// TwinCAT 3 PLC project Galimberti
// ProgramVersion: 3.1.4022.1
// libraries:
//   Tc2_MC2, * (Beckhoff Automation GmbH)
//   Tc2_MC2_Drive, * (Beckhoff Automation GmbH)
//   Tc2_Standard, * (Beckhoff Automation GmbH)
//   Tc2_System, * (Beckhoff Automation GmbH)
//   Tc3_Module, * (Beckhoff Automation GmbH)
// project tree:
//   DUTs/EVACUAZIONE SCARTI/ ES_ACTVAL.TcDUT, ES_MPO1.TcDUT, ES_PERSISTENT.TcDUT, ES_M.TcDUT, ES_ALARM.TcDUT, ES_S1.TcDUT, ES_S1PO1.TcDUT, ES_S2.TcDUT, ES_SEMAFORO.TcDUT, ES_T1.TcDUT, ES_T3.TcDUT, ES_T5.TcDUT, ES_T6.TcDUT
//   DUTs/RULLI_CENTRO_TAGLI/ dut_Axe_Status.TcDUT, dut_Dati_Pezzo.TcDUT
//   GVLs/EVACUAZIONE_SCARTI/ GVL_ES_IO.TcGVL
//   GVLs/RULLI CENTRO TAGLI/ GVL_CT_IO.TcGVL
//   / PlcTask.TcTTO, RulliCentroTagliTask.TcTTO
//   POUs/EVACUAZIONE_SCARTI/ EVACUAZIONE_SCARTI.TcPOU, MAIN.TcPOU
//   POUs/EVACUAZIONE_SCARTI/FB/ FB_AnalogSensor_full.TcPOU, FB_MMSensor_full.TcPOU, FB_Semaforo.TcPOU, fun_AreaM_SPEGNITUTTO.TcPOU
//   POUs/RULLI_CENTRO_TAGLI/FB/ FB_In_Position.TcPOU
//   POUs/RULLI_CENTRO_TAGLI/ MAIN_RCT.TcPOU, RULLI_CENTRO_TAGLI.TcPOU (not stored)
// real-time tasks:
//   TASK PlcTask: cycle T#10ms, priority 20, ADS port 350
//   TASK RulliCentroTagliTask: cycle T#10ms, priority 21, ADS port 351
// motion (NC):
//   TASK NC-Task 1 SAF: cycle T#2ms, priority 4, ADS port 501
//   TASK NC-Task 1 SVB: cycle T#10ms, priority 8, ADS port 511
//   AXIS C2M1 (id 1) // Motore catena 2
//     Dynamic: AccelerationMaximum=7500, DecelerationMaximum=7500, Acceleration=632.095593828125, Deceleration=632.095593828125, Jerk=1896.28678148437
//     Velo: RefSearch=4.21397062552083, RefSync=4.21397062552083, SlowManual=21.0698531276042, FastManual=126.419118765625, Fast=421.397062552083, Maximum=421.397062552083
//     OtherSettings: AllowMotionCmdToSlave=true
//     encoder EncType=8
//       EncPara: ScaleFactorNumerator=4.8964, ScaleFactorDenominator=1048576, MaxCount=#xffffffff
//     drive DrvType=9
//       DrvPara: MaxCount=#xffffffff, DriveControlDWord=#x00030100
//         Analog: VeloReferenz=463.536768807292, VeloScale=1.02400649589962, ScaleFactorActTorque=0.1
//         TimeComp: TaskDelayCycles=1
//     controller CtrType=1
//       CtrPara: PriorControlFactor=1
//         PosDiffControl: Range=30, Time=1
//         PID: PosKp=1.5
//         Observer: BandWidth=20
//   AXIS R1M1 (id 2) // Motore rulliera 1
//     Dynamic: Acceleration=1173.61, Deceleration=1173.61, Jerk=3520.84
//     Velo: RefSearch=7.8240862486901, RefSync=7.8240862486901, SlowManual=39.1204312434505, FastManual=234.722587460703, Fast=782.40862486901, Maximum=782.409
//     OtherSettings: AllowMotionCmdToSlave=true
//     encoder EncType=8
//       EncPara: ScaleFactorNumerator=9.091154, ScaleFactorDenominator=1048576, MaxCount=#xffffffff
//     drive DrvType=9
//       DrvPara: MaxCount=#xffffffff, DriveControlDWord=#x00030100
//         Analog: VeloReferenz=860.649487355912, VeloScale=1.02400649589962, ScaleFactorActTorque=0.1
//         TimeComp: TaskDelayCycles=1
//     controller CtrType=1
//       CtrPara: PriorControlFactor=1
//         Observer: BandWidth=20
//   AXIS C1M1 (id 3) // Motore sollevamento catenaria 1
//     Dynamic: Acceleration=194.243, Deceleration=194.243, Jerk=282.73
//     Velo: RefSearch=0.628289305598145, RefSync=0.628289305598145, SlowManual=3.14144652799072, FastManual=18.8486791679443, Fast=62.8289305598145, Maximum=62.8289
//     OtherSettings: AllowMotionCmdToSlave=true
//     encoder EncType=8
//       EncPara: ScaleFactorNumerator=1.15714, ScaleFactorDenominator=1048576, Inverse=true, MaxCount=#xffffffff
//         SoftEndMinControl: Enable=true, Range=590
//         SoftEndMaxControl: Enable=true, Range=1240
//     drive DrvType=9
//       DrvPara: Inverse=true, MaxCount=#xffffffff, DriveControlDWord=#x00030100
//         Analog: VeloReferenz=69.1118236157959, VeloScale=1.02400649589962, ScaleFactorActTorque=0.1
//         TimeComp: TaskDelayCycles=1
//     controller CtrType=1
//       CtrPara: PriorControlFactor=1
//         Observer: BandWidth=20
//   AXIS C1M3 (id 4) // Morore catenaria C1
//     Dynamic: AccelerationMaximum=7500, DecelerationMaximum=7500, Acceleration=900, Deceleration=900, Jerk=1896.28678148437
//     Velo: RefSearch=4.21397062552083, RefSync=4.21397062552083, SlowManual=21.0698531276042, FastManual=126.419118765625, Fast=421.397062552083, Maximum=421.397062552083
//     OtherSettings: AllowMotionCmdToSlave=true
//     encoder EncType=8
//       EncPara: ScaleFactorNumerator=4.8964, ScaleFactorDenominator=1048576, MaxCount=#xffffffff
//     drive DrvType=9
//       DrvPara: MaxCount=#xffffffff, DriveControlDWord=#x00030100
//         Analog: VeloReferenz=463.536768807292, VeloScale=1.02400649589962, ScaleFactorActTorque=0.1
//         TimeComp: TaskDelayCycles=1
//     controller CtrType=1
//       CtrPara: PriorControlFactor=1
//         PosDiffControl: Range=100, Time=1
//         PID: PosKp=2
//         Observer: BandWidth=20
//   AXIS C1M2 (id 5) // Rotazione catenaria C1
//     Dynamic: Acceleration=60.2372, Deceleration=60.2372, Jerk=180.712
//     Velo: RefSearch=0.401581141946615, RefSync=0.401581141946615, SlowManual=2.00790570973307, FastManual=12.0474342583984, Fast=40.1581141946615, Maximum=40.1581
//     OtherSettings: AllowMotionCmdToSlave=true
//     encoder EncType=8
//       EncPara: ScaleFactorNumerator=0.466615, ScaleFactorDenominator=1048576, MaxCount=#xffffffff
//     drive DrvType=9
//       DrvPara: MaxCount=#xffffffff, DriveControlDWord=#x00030100
//         Analog: VeloReferenz=44.1739256141276, VeloScale=1.02400649589962, ScaleFactorActTorque=0.1
//         TimeComp: TaskDelayCycles=1
//     controller CtrType=1
//       CtrPara: PriorControlFactor=1
//         Observer: BandWidth=20
//   AXIS C3 (id 6) // Catenaria 3
//     Dynamic: AccelerationMaximum=7000, Acceleration=689.378450181641, Deceleration=689.378450181641, Jerk=2068.13535054492
//     Velo: RefSearch=4.59585633454427, RefSync=4.59585633454427, SlowManual=22.9792816727214, FastManual=137.875690036328, Fast=459.585633454427, Maximum=459.585633454427
//     OtherSettings: AllowMotionCmdToSlave=true
//     encoder EncType=8
//       EncPara: ScaleFactorNumerator=5.34013, ScaleFactorDenominator=1048576, Inverse=true, MaxCount=#xffffffff
//     drive DrvType=9
//       DrvPara: Inverse=true, MaxCount=#xffffffff, DriveControlDWord=#x00030100
//         Analog: VeloReferenz=505.54419679987, VeloScale=1.02400649589962, ScaleFactorActTorque=0.1
//         TimeComp: TaskDelayCycles=1
//     controller CtrType=1
//       CtrPara: PriorControlFactor=1
//         Observer: BandWidth=20
//   AXIS C5 (id 7) // Catenaria 5
//     Dynamic: AccelerationMaximum=7000, Acceleration=689.378450181641, Deceleration=689.378450181641, Jerk=2068.13535054492
//     Velo: RefSearch=4.59585633454427, RefSync=4.59585633454427, SlowManual=22.9792816727214, FastManual=137.875690036328, Fast=459.585633454427, Maximum=459.585633454427
//     OtherSettings: AllowMotionCmdToSlave=true
//     encoder EncType=8
//       EncPara: ScaleFactorNumerator=5.34013, ScaleFactorDenominator=1048576, MaxCount=#xffffffff
//     drive DrvType=9
//       DrvPara: MaxCount=#xffffffff, DriveControlDWord=#x00030100
//         Analog: VeloReferenz=505.54419679987, VeloScale=1.02400649589962, ScaleFactorActTorque=0.1
//         TimeComp: TaskDelayCycles=1
//     controller CtrType=1
//       CtrPara: PriorControlFactor=1
//         Observer: BandWidth=20
//   AXIS C6 (id 8) // Catenaria 6
//     Dynamic: AccelerationMaximum=7000, Acceleration=689.378450181641, Deceleration=689.378450181641, Jerk=2068.13535054492
//     Velo: RefSearch=4.59585633454427, RefSync=4.59585633454427, SlowManual=22.9792816727214, FastManual=137.875690036328, Fast=459.585633454427, Maximum=459.585633454427
//     OtherSettings: AllowMotionCmdToSlave=true
//     encoder EncType=8
//       EncPara: ScaleFactorNumerator=5.34013, ScaleFactorDenominator=1048576, Inverse=true, MaxCount=#xffffffff
//     drive DrvType=9
//       DrvPara: Inverse=true, MaxCount=#xffffffff, DriveControlDWord=#x00030100
//         Analog: VeloReferenz=505.54419679987, VeloScale=1.02400649589962, ScaleFactorActTorque=0.1
//         TimeComp: TaskDelayCycles=1
//     controller CtrType=1
//       CtrPara: PriorControlFactor=1
//         Observer: BandWidth=20
//   AXIS R3 (id 9)
//     Dynamic: Acceleration=1353.648128, Deceleration=1353.648128, Jerk=4060.944384
//     Velo: RefSearch=9.02432085333333, RefSync=9.02432085333333, SlowManual=45.1216042666667, FastManual=270.7296256, Fast=902.432085333333, Maximum=902.432085333333
//     OtherSettings: AllowMotionCmdToSlave=true
//     encoder EncType=8
//       EncPara: ScaleFactorNumerator=10.48576, ScaleFactorDenominator=1048576, MaxCount=#xffffffff
//     drive DrvType=9
//       DrvPara: MaxCount=#xffffffff, DriveControlDWord=#x00030100
//         Analog: VeloReferenz=992.675293866667, VeloScale=1.02400649589962, ScaleFactorActTorque=0.1
//         TimeComp: TaskDelayCycles=1
//     controller CtrType=1
//       CtrPara: PriorControlFactor=1
//         Observer: BandWidth=20
//   AXIS R2 (id 10) // Rulliera 2
//     Dynamic: Acceleration=1173.61293730352, Deceleration=1173.61293730352, Jerk=3520.83881191055
//     Velo: RefSearch=7.8240862486901, RefSync=7.8240862486901, SlowManual=39.1204312434505, FastManual=234.722587460703, Fast=782.40862486901, Maximum=782.40862486901
//     OtherSettings: AllowMotionCmdToSlave=true
//     encoder EncType=8
//       EncPara: ScaleFactorNumerator=9.091154, ScaleFactorDenominator=1048576, MaxCount=#xffffffff
//     drive DrvType=9
//       DrvPara: MaxCount=#xffffffff, DriveControlDWord=#x00030100
//         Analog: VeloReferenz=860.649487355912, VeloScale=1.02400649589962, ScaleFactorActTorque=0.1
//         TimeComp: TaskDelayCycles=1
//     controller CtrType=1
//       CtrPara: PriorControlFactor=1
//         Observer: BandWidth=20
//   AXIS C4 (id 11)
//     Dynamic: AccelerationMaximum=7000, Acceleration=689.378450181641, Deceleration=689.378450181641, Jerk=2068.13535054492
//     Velo: RefSearch=4.59585633454427, RefSync=4.59585633454427, SlowManual=22.9792816727214, FastManual=137.875690036328, Fast=459.585633454427, Maximum=459.585633454427
//     OtherSettings: AllowMotionCmdToSlave=true
//     encoder EncType=8
//       EncPara: ScaleFactorNumerator=5.34013, ScaleFactorDenominator=1048576, MaxCount=#xffffffff
//     drive DrvType=9
//       DrvPara: MaxCount=#xffffffff, DriveControlDWord=#x00030100
//         Analog: VeloReferenz=505.54419679987, VeloScale=1.02400649589962, ScaleFactorActTorque=0.1
//         TimeComp: TaskDelayCycles=1
//     controller CtrType=1
//       CtrPara: PriorControlFactor=1
//         Observer: BandWidth=20
// I/O:
//   DEVICE Device 1 (EtherCAT), AmsNetId 192.168.30.180.2.1
//     Term 1 (EK1200) H-Q3 [EK1200-5000 EtherCAT Power supply (2A E-Bus)]
//       Term 2 (EL1008) [EL1008 8Ch. Dig. Input 24V, 3ms]
//       Term 3 (EL2008) [EL2008 8Ch. Dig. Output 24V, 0.5A]
//       Term 4 (EL6910) [EL6910, TwinSAFE PLC]
//       Term 5 (EK1110) [EK1110 EtherCAT extension]
//     Term 6 (EK1100) H-Q1 [EK1100 EtherCAT Coupler (2A E-Bus)]
//       Term 7 (EL1008) [EL1008 8Ch. Dig. Input 24V, 3ms]
//       Term 8 (EL1008) [EL1008 8Ch. Dig. Input 24V, 3ms]
//       Term 9 (EL2008) [EL2008 8Ch. Dig. Output 24V, 0.5A]
//       Term 10 (EL2008) [EL2008 8Ch. Dig. Output 24V, 0.5A]
//       Term 11 (EL3012) [EL3012 2Ch. Ana. Input 0-20mA DIFF]
//       Term 12 (EL3012) [EL3012 2Ch. Ana. Input 0-20mA DIFF]
//       Term 13 (EL2904) [EL2904, 4 Ch. Safety Output 24V, 0.5A, TwinSAFE]
//         modules: Module 1 (FSOES), Module 2 (DO)
//       Term 14 (EL2904) [EL2904, 4 Ch. Safety Output 24V, 0.5A, TwinSAFE]
//         modules: Module 1 (FSOES), Module 2 (DO)
//       Term 35 (EL6695) [EL6695 EtherCAT Bridge terminal (Primary)]
//       Term 15 (EK1110) [EK1110 EtherCAT extension]
//     Box 16 (EP6228-0022) M-CS1 [EP6228-0022 (IO Link Master)]
//       modules: Module 0 (DeviceState Inputs Device), Module 0 (DeviceState Inputs), Module 3 (IO-Link Slave) T1_SO1, Module 4 (empty), Module 5 (empty), Module 6 (empty), Module 7 (empty), Module 8 (empty), Module 9 (empty), Module 10 (empty)
//     Box 17 (EP6228-0022) T3-C01 [EP6228-0022 (IO Link Master)]
//       modules: Module 0 (DeviceState Inputs Device), Module 0 (DeviceState Inputs), Module 3 (IO-Link Slave), Module 2 (IO-Link Slave) S1_SO2, Module 3 (IO-Link Slave) S1_PO1, Module 6 (empty), Module 5 (IO-Link Slave) S1_Se1, Module 8 (empty), Module 7 (IO-Link Slave) T5_S1, Module 8 (IO-Link Slave) T5_SO1
//     Box 18 (EP1908) FS1 [EP1908, 8 Ch. Safety Input 24V, TwinSAFE]
//       modules: Module 1 (FSOE)
//     Term 39 (EK1100) [EK1100 EtherCAT Coupler (2A E-Bus)]
//       Term 40 (EL1008) [EL1008 8Ch. Dig. Input 24V, 3ms]
//       Term 41 (EL2008) [EL2008 8Ch. Dig. Output 24V, 0.5A]
//       Term 42 (EL2904) [EL2904, 4 Ch. Safety Output 24V, 0.5A, TwinSAFE]
//         modules: Module 1 (FSOES), Module 2 (DO)
//       Term 43 (EL1904) [EL1904, 4 Ch. Safety Input 24V, TwinSAFE]
//         modules: Module 1 (FSOES)
//       Term 44 (EL1904) [EL1904, 4 Ch. Safety Input 24V, TwinSAFE]
//         modules: Module 1 (FSOES)
//       Term 45 (EL1904) [EL1904, 4 Ch. Safety Input 24V, TwinSAFE]
//         modules: Module 1 (FSOES)
//       Term 46 (EK1122) [EK1122 2 port EtherCAT junction]
//         Box 47 (EP1008-0022) C1_CD4 [EP1008-0022 8 Ch. Dig. Input 24V, 3ms, M12]
//         Box 48 (EP6224-2022) C1_CO2 [EP6224-2022 (IO Link Master)]
//           modules: Module 1 (DeviceState Inputs Device), Module 2 (DeviceState Inputs), Module 3 (IO-Link Slave), Module 4 (IO-Link Slave), Module 5 (empty), Module 6 (empty)
//         Box 49 (EP1008-0022) C1_CD3 [EP1008-0022 8 Ch. Dig. Input 24V, 3ms, M12]
//         Box 50 (EP6224-2022) C1_CO1 [EP6224-2022 (IO Link Master)]
//           modules: Module 1 (DeviceState Inputs Device), Module 2 (DeviceState Inputs), Module 3 (IO-Link Slave), Module 4 (IO-Link Slave), Module 5 (IO-Link Slave), Module 6 (IO-Link Slave)
//         Box 51 (EP1008-0022) C1_CD2 [EP1008-0022 8 Ch. Dig. Input 24V, 3ms, M12]
//         Box 52 (EP1008-0022) C1_CD1 [EP1008-0022 8 Ch. Dig. Input 24V, 3ms, M12]
//         Box 53 (EP1008-0022) C2_CD4 [EP1008-0022 8 Ch. Dig. Input 24V, 3ms, M12]
//         Box 54 (EP6228-0022) C2_CO1 [EP6228-0022 (IO Link Master)]
//           modules: Module 1 (DeviceState Inputs Device), Module 2 (DeviceState Inputs), Module 3 (IO-Link Slave), Module 4 (IO-Link Slave), Module 5 (IO-Link Slave), Module 6 (IO-Link Slave), Module 7 (IO-Link Slave), Module 8 (IO-Link Slave), Module 9 (IO-Link Slave) - R1P5, Module 10 (IO-Link Slave) - R1P6
//         Box 55 (EP1008-0022) C2_CD3 [EP1008-0022 8 Ch. Dig. Input 24V, 3ms, M12]
//         Box 56 (EP1008-0022) C2_CD2 [EP1008-0022 8 Ch. Dig. Input 24V, 3ms, M12]
//         Box 57 (EP1008-0022) C2_CD1 [EP1008-0022 8 Ch. Dig. Input 24V, 3ms, M12]
//         Box 58 (EP6228-0022) C2_CO2 [EP6228-0022 (IO Link Master)]
//           modules: Module 1 (DeviceState Inputs Device), Module 2 (DeviceState Inputs), Module 3 (empty), Module 4 (IO-Link Slave) C1P1, Module 5 (empty), Module 6 (IO-Link Slave) R1P1, Module 7 (IO-Link Slave) R1P2, Module 8 (IO-Link Slave) R1P3, Module 9 (IO-Link Slave) R1P4, Module 10 (IO-Link Slave)
//         Box 59 (EP1908) C2_CS1 [EP1908, 8 Ch. Safety Input 24V, TwinSAFE]
//           modules: Module 1 (FSOE)
//         Box 60 (EP1908) C2_CS2 [EP1908, 8 Ch. Safety Input 24V, TwinSAFE]
//           modules: Module 1 (FSOE)
//       Term 61 (EK1122) [EK1122 2 port EtherCAT junction]
//         Drive 62 (AX5206-0000-0203) R2-C4 [AX5206-0000-0203 EtherCAT Drive (SoE, 2 Ch.)]
//         Drive 63 (AX5206-0000-0203) C3-R3 [AX5206-0000-0203 EtherCAT Drive (SoE, 2 Ch.)]
//         Drive 64 (AX5206-0000-0203) C5-C6 [AX5206-0000-0203 EtherCAT Drive (SoE, 2 Ch.)]
//         Drive 65 (AX5206-0000-0203) C1M2-C1M3 [AX5206-0000-0203 EtherCAT Drive (SoE, 2 Ch.)]
//         Drive 66 (AX5206-0000-0203) C2M1-R1M1 [AX5206-0000-0203 EtherCAT Drive (SoE, 2 Ch.)]
//         Drive 67 (AX5206-0000-0203) C1M1 [AX5112-0000-0203 EtherCAT Drive (SoE, 1 Ch.)]
//         Box 68 (S100) R1M2 [S100]
//         Box 99 (S100) R2 [S100]
//         Box 100 (S100) R3 [S100]
//         Box 101 (EP6228-0022) C5_CO1 [EP6228-0022 (IO Link Master)]
//           modules: Module 1 (DeviceState Inputs Device), Module 2 (DeviceState Inputs), Module 3 (IO-Link Slave), Module 4 (IO-Link Slave), Module 5 (IO-Link Slave), Module 6 (empty), Module 7 (IO-Link Slave), Module 8 (IO-Link Slave), Module 9 (IO-Link Slave), Module 10 (empty)
//         Box 102 (EP1008-0022) C5_CD1 [EP1008-0022 8 Ch. Dig. Input 24V, 3ms, M12]
//         Box 103 (EP1908) C5_CS1 [EP1908, 8 Ch. Safety Input 24V, TwinSAFE]
//           modules: Module 1 (FSOE)
//         Box 104 (EP6228-0022) C5_CO2 [EP6228-0022 (IO Link Master)]
//           modules: Module 1 (DeviceState Inputs Device), Module 2 (DeviceState Inputs), Module 3 (IO-Link Slave), Module 4 (IO-Link Slave), Module 5 (IO-Link Slave), Module 6 (IO-Link Slave), Module 7 (IO-Link Slave), Module 8 (IO-Link Slave), Module 9 (IO-Link Slave), Module 10 (IO-Link Slave)
//         Box 105 (EP1008-0022) C5_CD2 [EP1008-0022 8 Ch. Dig. Input 24V, 3ms, M12]
//         Box 106 (EP1008-0022) C5_CD3 [EP1008-0022 8 Ch. Dig. Input 24V, 3ms, M12]
//         Box 115 (EP1008-0022) C3CD1 [EP1008-0022 8 Ch. Dig. Input 24V, 3ms, M12]
//         Box 116 (EP6228-0022) C3CO1 [EP6228-0022 (IO Link Master)]
//           modules: Module 1 (DeviceState Inputs Device), Module 2 (DeviceState Inputs), Module 3 (empty), Module 4 (IO-Link Slave), Module 5 (IO-Link Slave), Module 6 (empty), Module 7 (empty), Module 8 (IO-Link Slave), Module 9 (IO-Link Slave), Module 10 (IO-Link Slave)
//         Box 117 (EP1008-0022) C3CD2 [EP1008-0022 8 Ch. Dig. Input 24V, 3ms, M12]
//         Box 118 (EP1908) C3CS1 [EP1908, 8 Ch. Safety Input 24V, TwinSAFE]
//           modules: Module 1 (FSOE)
//   DEVICE Device 4 (RT-Ethernet Protocol) (disabled), AmsNetId 192.168.30.180.5.1
//   DEVICE Device 5 (NOV-DP-RAM) (disabled)
// variable links:
//   Device 1 (EtherCAT) <-> Device 1 (EtherCAT)/Box 18 (EP1908) FS1
//     Term 1 (EK1200) H-Q3/Term 4 (EL6910)/ConnectionOutputs/TwinSafeGroup_ES.Box 18 (EP1908) - Module 1 (FSOE)_10 RxPDO <-> Module 1 (FSOE)/FSOE Inputs/FSOE
//   Device 1 (EtherCAT) <-> Device 1 (EtherCAT)/Term 1 (EK1200) H-Q3/Term 4 (EL6910)
//     Box 18 (EP1908) FS1/Module 1 (FSOE)/FSOE Outputs/FSOE <-> ConnectionInputs/TwinSafeGroup_ES.Box 18 (EP1908) - Module 1 (FSOE)_10 TxPDO
//     Term 39 (EK1100)/Term 42 (EL2904)/Module 1 (FSOES)/TxPDO/FSOE <-> ConnectionOutputs/TwinSafeGroup_ES.Term 42 (EL2904) - Module 1 (FSOES)_31 RxPDO
//     Term 39 (EK1100)/Term 44 (EL1904)/Module 1 (FSOES)/TxPDO/FSOE <-> ConnectionOutputs/TwinSafeGroup_ES.Term 44 (EL1904) - Module 1 (FSOES)_33 RxPDO
//     Term 39 (EK1100)/Term 43 (EL1904)/Module 1 (FSOES)/RxPDO/FSOE <-> ConnectionInputs/TwinSafeGroup_ES.Term 43 (EL1904) - Module 1 (FSOES)_32 TxPDO
//     Term 39 (EK1100)/Term 44 (EL1904)/Module 1 (FSOES)/RxPDO/FSOE <-> ConnectionInputs/TwinSafeGroup_ES.Term 44 (EL1904) - Module 1 (FSOES)_33 TxPDO
//     Term 39 (EK1100)/Term 46 (EK1122)/Box 59 (EP1908) C2_CS1/Module 1 (FSOE)/FSOE Inputs/FSOE <-> ConnectionOutputs/TwinSafeGroup_ES.Box 59 (EP1908) C2_CS1 - Module 1 (FSOE)_35 RxPDO
//     Term 39 (EK1100)/Term 46 (EK1122)/Box 60 (EP1908) C2_CS2/Module 1 (FSOE)/FSOE Inputs/FSOE <-> ConnectionOutputs/TwinSafeGroup_ES.Box 60 (EP1908) C2_CS2 - Module 1 (FSOE)_36 RxPDO
//     Term 39 (EK1100)/Term 46 (EK1122)/Box 59 (EP1908) C2_CS1/Module 1 (FSOE)/FSOE Outputs/FSOE <-> ConnectionInputs/TwinSafeGroup_ES.Box 59 (EP1908) C2_CS1 - Module 1 (FSOE)_35 TxPDO
//     Term 39 (EK1100)/Term 61 (EK1122)/Box 118 (EP1908) C3CS1/Module 1 (FSOE)/FSOE Inputs/FSOE <-> ConnectionOutputs/TwinSafeGroup_ES.Box 118 (EP1908) C3CS1 - Module 1 (FSOE)_39 RxPDO
//     Term 39 (EK1100)/Term 61 (EK1122)/Box 118 (EP1908) C3CS1/Module 1 (FSOE)/FSOE Outputs/FSOE <-> ConnectionInputs/TwinSafeGroup_ES.Box 118 (EP1908) C3CS1 - Module 1 (FSOE)_39 TxPDO
//     Term 6 (EK1100) H-Q1/Term 13 (EL2904)/Module 1 (FSOES)/TxPDO/FSOE <-> ConnectionOutputs/TwinSafeGroup_ES.Term 13 (EL2904) - Module 1 (FSOES)_8 RxPDO
//   Device 1 (EtherCAT) <-> Device 1 (EtherCAT)/Term 39 (EK1100)/Term 42 (EL2904)
//     Term 1 (EK1200) H-Q3/Term 4 (EL6910)/ConnectionInputs/TwinSafeGroup_ES.Term 42 (EL2904) - Module 1 (FSOES)_31 TxPDO <-> Module 1 (FSOES)/RxPDO/FSOE
//   Device 1 (EtherCAT) <-> Device 1 (EtherCAT)/Term 39 (EK1100)/Term 43 (EL1904)
//     Term 1 (EK1200) H-Q3/Term 4 (EL6910)/ConnectionOutputs/TwinSafeGroup_ES.Term 43 (EL1904) - Module 1 (FSOES)_32 RxPDO <-> Module 1 (FSOES)/TxPDO/FSOE
//   Device 1 (EtherCAT) <-> Device 1 (EtherCAT)/Term 39 (EK1100)/Term 45 (EL1904)
//     Term 1 (EK1200) H-Q3/Term 4 (EL6910)/ConnectionInputs/TwinSafeGroup_ES.Term 45 (EL1904) - Module 1 (FSOES)_34 TxPDO <-> Module 1 (FSOES)/RxPDO/FSOE
//     Term 1 (EK1200) H-Q3/Term 4 (EL6910)/ConnectionOutputs/TwinSafeGroup_ES.Term 45 (EL1904) - Module 1 (FSOES)_34 RxPDO <-> Module 1 (FSOES)/TxPDO/FSOE
//   Device 1 (EtherCAT) <-> Device 1 (EtherCAT)/Term 39 (EK1100)/Term 46 (EK1122)/Box 60 (EP1908) C2_CS2
//     Term 1 (EK1200) H-Q3/Term 4 (EL6910)/ConnectionInputs/TwinSafeGroup_ES.Box 60 (EP1908) C2_CS2 - Module 1 (FSOE)_36 TxPDO <-> Module 1 (FSOE)/FSOE Outputs/FSOE
//   Device 1 (EtherCAT) <-> Device 1 (EtherCAT)/Term 39 (EK1100)/Term 61 (EK1122)/Box 103 (EP1908) C5_CS1
//     Term 1 (EK1200) H-Q3/Term 4 (EL6910)/ConnectionInputs/TwinSafeGroup_ES.Box 103 (EP1908) C5_CS1 - Module 1 (FSOE)_40 TxPDO <-> Module 1 (FSOE)/FSOE Outputs/FSOE
//     Term 1 (EK1200) H-Q3/Term 4 (EL6910)/ConnectionOutputs/TwinSafeGroup_ES.Box 103 (EP1908) C5_CS1 - Module 1 (FSOE)_40 RxPDO <-> Module 1 (FSOE)/FSOE Inputs/FSOE
//   Device 1 (EtherCAT) <-> Device 1 (EtherCAT)/Term 6 (EK1100) H-Q1/Term 13 (EL2904)
//     Term 1 (EK1200) H-Q3/Term 4 (EL6910)/ConnectionInputs/TwinSafeGroup_ES.Term 13 (EL2904) - Module 1 (FSOES)_8 TxPDO <-> Module 1 (FSOES)/RxPDO/FSOE
//   NC-Task 1 SAF/Axes/C1M1 <-> Device 1 (EtherCAT)/Term 39 (EK1100)/Term 61 (EK1122)/Drive 67 (AX5206-0000-0203) C1M1
//     Drive/Inputs/In/nDataIn1 <-> AT/Following distance
//     Drive/Inputs/In/nDcOutputTime <-> InfoData/DcOutputShift
//     Drive/Inputs/In/nState1 <-> AT/Drive status word @bit 8
//     Drive/Inputs/In/nState2 <-> AT/Drive status word
//     Drive/Inputs/In/nState4 @bit 1 <-> WcState/InputToggle
//     Drive/Inputs/In/nState4 <-> WcState/WcState
//     Drive/Outputs/Out/nCtrl1 <-> MDT/Master control word @bit 8
//     Drive/Outputs/Out/nDataOut1 <-> MDT/Position command value
//     Enc/Inputs/In/nDataIn1 <-> AT/Position feedback 1 value
//     Enc/Inputs/In/nDcInputTime <-> InfoData/DcInputShift
//     Enc/Inputs/In/nState4 @bit 1 <-> WcState/InputToggle
//     Enc/Inputs/In/nState4 <-> WcState/WcState
//   NC-Task 1 SAF/Axes/C1M2 <-> Device 1 (EtherCAT)/Term 39 (EK1100)/Term 61 (EK1122)/Drive 65 (AX5206-0000-0203) C1M2-C1M3
//     Drive/Inputs/In/nDataIn1 <-> AT 1/Following distance
//     Drive/Inputs/In/nDataIn3[0] <-> AT 1/Torque feedback value
//     Drive/Inputs/In/nDcOutputTime <-> InfoData/DcOutputShift
//     Drive/Inputs/In/nState1 <-> AT 1/Drive status word @bit 8
//     Drive/Inputs/In/nState2 <-> AT 1/Drive status word
//     Drive/Inputs/In/nState4 @bit 1 <-> WcState/InputToggle
//     Drive/Inputs/In/nState4 <-> WcState/WcState
//     Drive/Outputs/Out/nCtrl1 <-> MDT 1/Master control word @bit 8
//     Drive/Outputs/Out/nDataOut1 <-> MDT 1/Position command value
//     Enc/Inputs/In/nDataIn1 <-> AT 1/Position feedback 1 value
//     Enc/Inputs/In/nDcInputTime <-> InfoData/DcInputShift
//     Enc/Inputs/In/nState4 @bit 1 <-> WcState/InputToggle
//     Enc/Inputs/In/nState4 <-> WcState/WcState
//   NC-Task 1 SAF/Axes/C1M3 <-> Device 1 (EtherCAT)/Term 39 (EK1100)/Term 61 (EK1122)/Drive 65 (AX5206-0000-0203) C1M2-C1M3
//     Drive/Inputs/In/nDataIn1 <-> AT 2/Following distance
//     Drive/Inputs/In/nDcOutputTime <-> InfoData/DcOutputShift
//     Drive/Inputs/In/nState1 <-> AT 2/Drive status word @bit 8
//     Drive/Inputs/In/nState2 <-> AT 2/Drive status word
//     Drive/Inputs/In/nState4 @bit 1 <-> WcState/InputToggle
//     Drive/Inputs/In/nState4 <-> WcState/WcState
//     Drive/Outputs/Out/nCtrl1 <-> MDT 2/Master control word @bit 8
//     Drive/Outputs/Out/nDataOut1 <-> MDT 2/Position command value
//     Enc/Inputs/In/nDataIn1 <-> AT 2/Position feedback 1 value
//     Enc/Inputs/In/nDcInputTime <-> InfoData/DcInputShift
//     Enc/Inputs/In/nState4 @bit 1 <-> WcState/InputToggle
//     Enc/Inputs/In/nState4 <-> WcState/WcState
//   NC-Task 1 SAF/Axes/C2M1 <-> Device 1 (EtherCAT)/Term 39 (EK1100)/Term 61 (EK1122)/Drive 66 (AX5206-0000-0203) C2M1-R1M1
//     Drive/Inputs/In/nDataIn1 <-> AT 1/Following distance
//     Drive/Inputs/In/nDcOutputTime <-> InfoData/DcOutputShift
//     Drive/Inputs/In/nState1 <-> AT 1/Drive status word @bit 8
//     Drive/Inputs/In/nState2 <-> AT 1/Drive status word
//     Drive/Inputs/In/nState4 @bit 1 <-> WcState/InputToggle
//     Drive/Inputs/In/nState4 <-> WcState/WcState
//     Drive/Outputs/Out/nCtrl1 <-> MDT 1/Master control word @bit 8
//     Drive/Outputs/Out/nDataOut1 <-> MDT 1/Position command value
//     Enc/Inputs/In/nDataIn1 <-> AT 1/Position feedback 1 value
//     Enc/Inputs/In/nDcInputTime <-> InfoData/DcInputShift
//     Enc/Inputs/In/nState4 @bit 1 <-> WcState/InputToggle
//     Enc/Inputs/In/nState4 <-> WcState/WcState
//   NC-Task 1 SAF/Axes/C3 <-> Device 1 (EtherCAT)/Term 39 (EK1100)/Term 61 (EK1122)/Drive 63 (AX5206-0000-0203) C3-R3
//     Drive/Inputs/In/nDataIn1 <-> AT 1/Following distance
//     Drive/Inputs/In/nDcOutputTime <-> InfoData/DcOutputShift
//     Drive/Inputs/In/nState1 <-> AT 1/Drive status word @bit 8
//     Drive/Inputs/In/nState2 <-> AT 1/Drive status word
//     Drive/Inputs/In/nState4 @bit 1 <-> WcState/InputToggle
//     Drive/Inputs/In/nState4 <-> WcState/WcState
//     Drive/Outputs/Out/nCtrl1 <-> MDT 1/Master control word @bit 8
//     Drive/Outputs/Out/nDataOut1 <-> MDT 1/Position command value
//     Enc/Inputs/In/nDataIn1 <-> AT 1/Position feedback 1 value
//     Enc/Inputs/In/nDcInputTime <-> InfoData/DcInputShift
//     Enc/Inputs/In/nState4 @bit 1 <-> WcState/InputToggle
//     Enc/Inputs/In/nState4 <-> WcState/WcState
//   NC-Task 1 SAF/Axes/C4 <-> Device 1 (EtherCAT)/Term 39 (EK1100)/Term 61 (EK1122)/Drive 62 (AX5206-0000-0203) R2-C4
//     Drive/Inputs/In/nDataIn1 <-> AT 2/Following distance
//     Drive/Inputs/In/nDcOutputTime <-> InfoData/DcOutputShift
//     Drive/Inputs/In/nState1 <-> AT 2/Drive status word @bit 8
//     Drive/Inputs/In/nState2 <-> AT 2/Drive status word
//     Drive/Inputs/In/nState4 @bit 1 <-> WcState/InputToggle
//     Drive/Inputs/In/nState4 <-> WcState/WcState
//     Drive/Outputs/Out/nCtrl1 <-> MDT 2/Master control word @bit 8
//     Drive/Outputs/Out/nDataOut1 <-> MDT 2/Position command value
//     Enc/Inputs/In/nDataIn1 <-> AT 2/Position feedback 1 value
//     Enc/Inputs/In/nDcInputTime <-> InfoData/DcInputShift
//     Enc/Inputs/In/nState4 @bit 1 <-> WcState/InputToggle
//     Enc/Inputs/In/nState4 <-> WcState/WcState
//   NC-Task 1 SAF/Axes/C5 <-> Device 1 (EtherCAT)/Term 39 (EK1100)/Term 61 (EK1122)/Drive 64 (AX5206-0000-0203) C5-C6
//     Drive/Inputs/In/nDataIn1 <-> AT 1/Following distance
//     Drive/Inputs/In/nDcOutputTime <-> InfoData/DcOutputShift
//     Drive/Inputs/In/nState1 <-> AT 1/Drive status word @bit 8
//     Drive/Inputs/In/nState2 <-> AT 1/Drive status word
//     Drive/Inputs/In/nState4 @bit 1 <-> WcState/InputToggle
//     Drive/Inputs/In/nState4 <-> WcState/WcState
//     Drive/Outputs/Out/nCtrl1 <-> MDT 1/Master control word @bit 8
//     Drive/Outputs/Out/nDataOut1 <-> MDT 1/Position command value
//     Enc/Inputs/In/nDataIn1 <-> AT 1/Position feedback 1 value
//     Enc/Inputs/In/nDcInputTime <-> InfoData/DcInputShift
//     Enc/Inputs/In/nState4 @bit 1 <-> WcState/InputToggle
//     Enc/Inputs/In/nState4 <-> WcState/WcState
//   NC-Task 1 SAF/Axes/C6 <-> Device 1 (EtherCAT)/Term 39 (EK1100)/Term 61 (EK1122)/Drive 64 (AX5206-0000-0203) C5-C6
//     Drive/Inputs/In/nDataIn1 <-> AT 2/Following distance
//     Drive/Inputs/In/nDcOutputTime <-> InfoData/DcOutputShift
//     Drive/Inputs/In/nState1 <-> AT 2/Drive status word @bit 8
//     Drive/Inputs/In/nState2 <-> AT 2/Drive status word
//     Drive/Inputs/In/nState4 @bit 1 <-> WcState/InputToggle
//     Drive/Inputs/In/nState4 <-> WcState/WcState
//     Drive/Outputs/Out/nCtrl1 <-> MDT 2/Master control word @bit 8
//     Drive/Outputs/Out/nDataOut1 <-> MDT 2/Position command value
//     Enc/Inputs/In/nDataIn1 <-> AT 2/Position feedback 1 value
//     Enc/Inputs/In/nDcInputTime <-> InfoData/DcInputShift
//     Enc/Inputs/In/nState4 @bit 1 <-> WcState/InputToggle
//     Enc/Inputs/In/nState4 <-> WcState/WcState
//   NC-Task 1 SAF/Axes/R1M1 <-> Device 1 (EtherCAT)/Term 39 (EK1100)/Term 61 (EK1122)/Drive 66 (AX5206-0000-0203) C2M1-R1M1
//     Drive/Inputs/In/nDataIn1 <-> AT 2/Following distance
//     Drive/Inputs/In/nDcOutputTime <-> InfoData/DcOutputShift
//     Drive/Inputs/In/nState1 <-> AT 2/Drive status word @bit 8
//     Drive/Inputs/In/nState2 <-> AT 2/Drive status word
//     Drive/Inputs/In/nState4 @bit 1 <-> WcState/InputToggle
//     Drive/Inputs/In/nState4 <-> WcState/WcState
//     Drive/Outputs/Out/nCtrl1 <-> MDT 2/Master control word @bit 8
//     Drive/Outputs/Out/nDataOut1 <-> MDT 2/Position command value
//     Enc/Inputs/In/nDataIn1 <-> AT 2/Position feedback 1 value
//     Enc/Inputs/In/nDcInputTime <-> InfoData/DcInputShift
//     Enc/Inputs/In/nState4 @bit 1 <-> WcState/InputToggle
//     Enc/Inputs/In/nState4 <-> WcState/WcState
//   NC-Task 1 SAF/Axes/R2 <-> Device 1 (EtherCAT)/Term 39 (EK1100)/Term 61 (EK1122)/Drive 62 (AX5206-0000-0203) R2-C4
//     Drive/Inputs/In/nDataIn1 <-> AT 1/Following distance
//     Drive/Inputs/In/nDcOutputTime <-> InfoData/DcOutputShift
//     Drive/Inputs/In/nState1 <-> AT 1/Drive status word @bit 8
//     Drive/Inputs/In/nState2 <-> AT 1/Drive status word
//     Drive/Inputs/In/nState4 @bit 1 <-> WcState/InputToggle
//     Drive/Inputs/In/nState4 <-> WcState/WcState
//     Drive/Outputs/Out/nCtrl1 <-> MDT 1/Master control word @bit 8
//     Drive/Outputs/Out/nDataOut1 <-> MDT 1/Position command value
//     Enc/Inputs/In/nDataIn1 <-> AT 1/Position feedback 1 value
//     Enc/Inputs/In/nDcInputTime <-> InfoData/DcInputShift
//     Enc/Inputs/In/nState4 @bit 1 <-> WcState/InputToggle
//     Enc/Inputs/In/nState4 <-> WcState/WcState
//   NC-Task 1 SAF/Axes/R3 <-> Device 1 (EtherCAT)/Term 39 (EK1100)/Term 61 (EK1122)/Drive 63 (AX5206-0000-0203) C3-R3
//     Drive/Inputs/In/nDataIn1 <-> AT 2/Following distance
//     Drive/Inputs/In/nDcOutputTime <-> InfoData/DcOutputShift
//     Drive/Inputs/In/nState1 <-> AT 2/Drive status word @bit 8
//     Drive/Inputs/In/nState2 <-> AT 2/Drive status word
//     Drive/Inputs/In/nState4 @bit 1 <-> WcState/InputToggle
//     Drive/Inputs/In/nState4 <-> WcState/WcState
//     Drive/Outputs/Out/nCtrl1 <-> MDT 2/Master control word @bit 8
//     Drive/Outputs/Out/nDataOut1 <-> MDT 2/Position command value
//     Enc/Inputs/In/nDataIn1 <-> AT 2/Position feedback 1 value
//     Enc/Inputs/In/nDcInputTime <-> InfoData/DcInputShift
//     Enc/Inputs/In/nState4 @bit 1 <-> WcState/InputToggle
//     Enc/Inputs/In/nState4 <-> WcState/WcState
//   Galimberti/Galimberti Instance <-> Device 1 (EtherCAT)/Box 16 (EP6228-0022) M-CS1
//     PlcTask Inputs/.glo_analog_in_MCS1[1] <-> Module 3 (IO-Link Slave) T1_SO1/IO-Link Port1/Distance
//     RulliCentroTagliTask Inputs/.glo_IOLState_MCS1[{1..8}] <-> Module 0 (DeviceState Inputs)/DeviceState Inputs/State Ch{1..8}  (8 links)
//     RulliCentroTagliTask Inputs/.glo_State_MCS1[1] <-> InfoData/State
//     RulliCentroTagliTask Inputs/.glo_WcState_MCS1[1] <-> WcState/WcState
//   Galimberti/Galimberti Instance <-> Device 1 (EtherCAT)/Box 17 (EP6228-0022) T3-C01
//     PlcTask Inputs/.glo_analog_in_T3C01[1] <-> Module 2 (IO-Link Slave) S1_SO2/IO-Link Port2/PDV1
//     PlcTask Inputs/.glo_analog_in_T3C01[2] <-> Module 8 (IO-Link Slave) T5_SO1/IO-Link Port8/PDV1
//     PlcTask Inputs/.glo_dig_in_T3C01[10] <-> Module 3 (IO-Link Slave)/IO-Link Port1/Port1: process data
//     PlcTask Inputs/.glo_dig_in_T3C01[1] <-> Module 3 (IO-Link Slave) S1_PO1/IO-Link Port3_in/Switchstate Pin 1 (Bit0.0)
//     PlcTask Inputs/.glo_dig_in_T3C01[2] <-> Module 3 (IO-Link Slave) S1_PO1/IO-Link Port3_in/Switchstate Pin 2 (Bit0.1)
//     PlcTask Inputs/.glo_dig_in_T3C01[3] <-> Module 3 (IO-Link Slave) S1_PO1/IO-Link Port3_in/Switchstate Pin 3 (Bit0.2)
//     PlcTask Inputs/.glo_dig_in_T3C01[4] <-> Module 3 (IO-Link Slave) S1_PO1/IO-Link Port3_in/Switchstate Pin 4 (Bit0.3)
//     PlcTask Inputs/.glo_dig_in_T3C01[5] <-> Module 3 (IO-Link Slave) S1_PO1/IO-Link Port3_in/Switchstate Pin 5 (Bit0.4)
//     PlcTask Inputs/.glo_dig_in_T3C01[6] <-> Module 3 (IO-Link Slave) S1_PO1/IO-Link Port3_in/Switchstate Pin 6 (Bit0.5)
//     PlcTask Inputs/.glo_dig_in_T3C01[7] <-> Module 3 (IO-Link Slave) S1_PO1/IO-Link Port3_in/Switchstate Pin 7 (Bit0.6)
//     PlcTask Inputs/.glo_dig_in_T3C01[8] <-> Module 3 (IO-Link Slave) S1_PO1/IO-Link Port3_in/Switchstate Pin 8 (Bit0.7)
//     PlcTask Inputs/.glo_dig_in_T3C01[25] <-> Module 7 (IO-Link Slave) T5_S1/IO-Link Port7/Port7: process data
//     PlcTask Outputs/.S1_Se1.analog{0..5} <-> Module 5 (IO-Link Slave) S1_Se1/IO-Link Port5/Port5: process data[{0..5}]  (6 links)
//     PlcTask Outputs/.glo_dig_out_T3C01[1] <-> Module 3 (IO-Link Slave) S1_PO1/IO-Link Port3_out/Switchstate Pin 1 (Bit0.0)
//     PlcTask Outputs/.glo_dig_out_T3C01[2] <-> Module 3 (IO-Link Slave) S1_PO1/IO-Link Port3_out/Switchstate Pin 2 (Bit0.1)
//     PlcTask Outputs/.glo_dig_out_T3C01[3] <-> Module 3 (IO-Link Slave) S1_PO1/IO-Link Port3_out/Switchstate Pin 3 (Bit0.2)
//     PlcTask Outputs/.glo_dig_out_T3C01[4] <-> Module 3 (IO-Link Slave) S1_PO1/IO-Link Port3_out/Switchstate Pin 4 (Bit0.3)
//     PlcTask Outputs/.glo_dig_out_T3C01[5] <-> Module 3 (IO-Link Slave) S1_PO1/IO-Link Port3_out/Switchstate Pin 5 (Bit0.4)
//     PlcTask Outputs/.glo_dig_out_T3C01[6] <-> Module 3 (IO-Link Slave) S1_PO1/IO-Link Port3_out/Switchstate Pin 6 (Bit0.5)
//     PlcTask Outputs/.glo_dig_out_T3C01[7] <-> Module 3 (IO-Link Slave) S1_PO1/IO-Link Port3_out/Switchstate Pin 7 (Bit0.6)
//     PlcTask Outputs/.glo_dig_out_T3C01[8] <-> Module 3 (IO-Link Slave) S1_PO1/IO-Link Port3_out/Switchstate Pin 8 (Bit0.7)
//     RulliCentroTagliTask Inputs/.glo_IOLState_T3C01[1] <-> Module 0 (DeviceState Inputs)/DeviceState Inputs/State Ch1
//     RulliCentroTagliTask Inputs/.glo_IOLState_T3C01[2] <-> Module 0 (DeviceState Inputs)/DeviceState Inputs/State Ch2
//     RulliCentroTagliTask Inputs/.glo_IOLState_T3C01[3] <-> Module 0 (DeviceState Inputs)/DeviceState Inputs/State Ch3
//     RulliCentroTagliTask Inputs/.glo_IOLState_T3C01[4] <-> Module 0 (DeviceState Inputs)/DeviceState Inputs/State Ch4
//     RulliCentroTagliTask Inputs/.glo_IOLState_T3C01[5] <-> Module 0 (DeviceState Inputs)/DeviceState Inputs/State Ch5
//     RulliCentroTagliTask Inputs/.glo_IOLState_T3C01[6] <-> Module 0 (DeviceState Inputs)/DeviceState Inputs/State Ch6
//     RulliCentroTagliTask Inputs/.glo_IOLState_T3C01[7] <-> Module 0 (DeviceState Inputs)/DeviceState Inputs/State Ch7
//     RulliCentroTagliTask Inputs/.glo_IOLState_T3C01[8] <-> Module 0 (DeviceState Inputs)/DeviceState Inputs/State Ch8
//     RulliCentroTagliTask Inputs/.glo_State_T3C01[1] <-> InfoData/State
//     RulliCentroTagliTask Inputs/.glo_WcState_T3C01[1] <-> WcState/WcState
//   Galimberti/Galimberti Instance <-> Device 1 (EtherCAT)/Term 1 (EK1200) H-Q3/Term 2 (EL1008)
//     RulliCentroTagliTask Inputs/.glo_State_HQ3[1] <-> InfoData/State
//     RulliCentroTagliTask Inputs/.glo_WcState_HQ3[1] <-> WcState/WcState
//     RulliCentroTagliTask Inputs/.glo_dig_in_HQ3[{1..8}] <-> Channel {1..8}/Input  (8 links)
//   Galimberti/Galimberti Instance <-> Device 1 (EtherCAT)/Term 1 (EK1200) H-Q3/Term 3 (EL2008)
//     RulliCentroTagliTask Inputs/.glo_State_HQ3[2] <-> InfoData/State
//     RulliCentroTagliTask Inputs/.glo_WcState_HQ3[2] <-> WcState/WcState
//     RulliCentroTagliTask Outputs/.glo_dig_out_HQ3[{1..8}] <-> Channel {1..8}/Output  (8 links)
//   Galimberti/Galimberti Instance <-> Device 1 (EtherCAT)/Term 1 (EK1200) H-Q3/Term 4 (EL6910)
//     PlcTask Inputs/.TS_AreaM_ON <-> StandardInputs/TwinSafeGroup_ES.toTC_AreaM_ON_23
//     PlcTask Inputs/.TS_AreaS_ON <-> StandardInputs/TwinSafeGroup_ES.toTC_AreaS_ON_24
//     PlcTask Outputs/.TS_ErrAck <-> StandardOutputs/TwinSafeGroup_ES.ErrorAcknowledgement_1
//     PlcTask Outputs/.TS_MPO1_Rst_Area_Macinatore <-> StandardOutputs/TwinSafeGroup_ES.fromTC_Rst_Area_Macinatore_43
//     PlcTask Outputs/.TS_Run_GrpES <-> StandardOutputs/TwinSafeGroup_ES.Run_2
//     PlcTask Outputs/.TS_S1PO1_btn_R <-> StandardOutputs/TwinSafeGroup_ES.fromTC_S1PO1_RestartE_stop_20
//     RulliCentroTagliTask Inputs/.TS_AreaM_OFF <-> StandardInputs/TwinSafeGroup_ES.toTC_AreaM_ON_23
//     RulliCentroTagliTask Inputs/.TS_ComErr <-> StandardInputs/TwinSafeGroup_ES.toTC_ComErr_27
//     RulliCentroTagliTask Inputs/.TS_FBErr <-> StandardInputs/TwinSafeGroup_ES.toTC_FBErr_28
//     RulliCentroTagliTask Inputs/.TS_R1P1_Pls_Eme <-> StandardInputs/TwinSafeGroup_ES.toTC_Eme_Ok_38
//     RulliCentroTagliTask Inputs/.TS_S1PO1_btn_Emerg <-> StandardInputs/TwinSafeGroup_ES.toTC_S1PO1_Emergency_21
//     RulliCentroTagliTask Inputs/.TS_S1PR1_Door <-> StandardInputs/TwinSafeGroup_ES.toTC_S1PR1_Door_22
//     RulliCentroTagliTask Inputs/.glo_State_HQ3[3] <-> InfoData/State
//     RulliCentroTagliTask Inputs/.glo_WcState_HQ3[3] <-> WcState/WcState
//     RulliCentroTagliTask Inputs/.glo_dig_in_BOX18[{1..8}] <-> Connection Info Data/TwinSafeGroup_ES.Box 18 (EP1908) - Module 1 (FSOE)_10 Info Data/Input Safe Data InputChannel{1..8}  (8 links)
//     RulliCentroTagliTask Inputs/.glo_dig_in_C2_CS1[1] <-> Connection Info Data/TwinSafeGroup_ES.Box 59 (EP1908) C2_CS1 - Module 1 (FSOE)_35 Info Data/Input Safe Data InputChannel1
//     RulliCentroTagliTask Inputs/.glo_dig_in_C2_CS1[2] <-> Connection Info Data/TwinSafeGroup_ES.Box 59 (EP1908) C2_CS1 - Module 1 (FSOE)_35 Info Data/Input Safe Data InputChannel2
//     RulliCentroTagliTask Inputs/.glo_dig_in_C2_CS1[3] <-> Connection Info Data/TwinSafeGroup_ES.Box 59 (EP1908) C2_CS1 - Module 1 (FSOE)_35 Info Data/Input Safe Data InputChannel3
//     RulliCentroTagliTask Inputs/.glo_dig_in_C2_CS1[4] <-> Connection Info Data/TwinSafeGroup_ES.Box 59 (EP1908) C2_CS1 - Module 1 (FSOE)_35 Info Data/Input Safe Data InputChannel4
//     RulliCentroTagliTask Inputs/.glo_dig_in_C2_CS1[5] <-> Connection Info Data/TwinSafeGroup_ES.Box 59 (EP1908) C2_CS1 - Module 1 (FSOE)_35 Info Data/Input Safe Data InputChannel5
//     RulliCentroTagliTask Inputs/.glo_dig_in_C2_CS1[6] <-> Connection Info Data/TwinSafeGroup_ES.Box 59 (EP1908) C2_CS1 - Module 1 (FSOE)_35 Info Data/Input Safe Data InputChannel6
//     RulliCentroTagliTask Inputs/.glo_dig_in_C2_CS1[7] <-> Connection Info Data/TwinSafeGroup_ES.Box 59 (EP1908) C2_CS1 - Module 1 (FSOE)_35 Info Data/Input Safe Data InputChannel7
//     RulliCentroTagliTask Inputs/.glo_dig_in_C2_CS1[8] <-> Connection Info Data/TwinSafeGroup_ES.Box 59 (EP1908) C2_CS1 - Module 1 (FSOE)_35 Info Data/Input Safe Data InputChannel8
//     RulliCentroTagliTask Inputs/.glo_dig_in_C2_CS2[1] <-> Connection Info Data/TwinSafeGroup_ES.Box 60 (EP1908) C2_CS2 - Module 1 (FSOE)_36 Info Data/Input Safe Data InputChannel1
//     RulliCentroTagliTask Inputs/.glo_dig_in_C2_CS2[2] <-> Connection Info Data/TwinSafeGroup_ES.Box 60 (EP1908) C2_CS2 - Module 1 (FSOE)_36 Info Data/Input Safe Data InputChannel2
//     RulliCentroTagliTask Inputs/.glo_dig_in_C2_CS2[3] <-> Connection Info Data/TwinSafeGroup_ES.Box 60 (EP1908) C2_CS2 - Module 1 (FSOE)_36 Info Data/Input Safe Data InputChannel3
//     RulliCentroTagliTask Inputs/.glo_dig_in_C2_CS2[4] <-> Connection Info Data/TwinSafeGroup_ES.Box 60 (EP1908) C2_CS2 - Module 1 (FSOE)_36 Info Data/Input Safe Data InputChannel4
//     RulliCentroTagliTask Inputs/.glo_dig_in_C2_CS2[5] <-> Connection Info Data/TwinSafeGroup_ES.Box 60 (EP1908) C2_CS2 - Module 1 (FSOE)_36 Info Data/Input Safe Data InputChannel5
//     RulliCentroTagliTask Inputs/.glo_dig_in_C2_CS2[6] <-> Connection Info Data/TwinSafeGroup_ES.Box 60 (EP1908) C2_CS2 - Module 1 (FSOE)_36 Info Data/Input Safe Data InputChannel6
//     RulliCentroTagliTask Inputs/.glo_dig_in_C2_CS2[7] <-> Connection Info Data/TwinSafeGroup_ES.Box 60 (EP1908) C2_CS2 - Module 1 (FSOE)_36 Info Data/Input Safe Data InputChannel7
//     RulliCentroTagliTask Inputs/.glo_dig_in_C2_CS2[8] <-> Connection Info Data/TwinSafeGroup_ES.Box 60 (EP1908) C2_CS2 - Module 1 (FSOE)_36 Info Data/Input Safe Data InputChannel8
//     RulliCentroTagliTask Inputs/.glo_dig_in_C5_CS1[1] <-> Connection Info Data/TwinSafeGroup_ES.Box 103 (EP1908) C5_CS1 - Module 1 (FSOE)_40 Info Data/Input Safe Data InputChannel1
//     RulliCentroTagliTask Inputs/.glo_dig_in_C5_CS1[2] <-> Connection Info Data/TwinSafeGroup_ES.Box 103 (EP1908) C5_CS1 - Module 1 (FSOE)_40 Info Data/Input Safe Data InputChannel2
//     RulliCentroTagliTask Inputs/.glo_dig_in_C5_CS1[3] <-> Connection Info Data/TwinSafeGroup_ES.Box 103 (EP1908) C5_CS1 - Module 1 (FSOE)_40 Info Data/Input Safe Data InputChannel3
//     RulliCentroTagliTask Inputs/.glo_dig_in_C5_CS1[4] <-> Connection Info Data/TwinSafeGroup_ES.Box 103 (EP1908) C5_CS1 - Module 1 (FSOE)_40 Info Data/Input Safe Data InputChannel4
//     RulliCentroTagliTask Inputs/.glo_dig_in_C5_CS1[5] <-> Connection Info Data/TwinSafeGroup_ES.Box 103 (EP1908) C5_CS1 - Module 1 (FSOE)_40 Info Data/Input Safe Data InputChannel5
//     RulliCentroTagliTask Inputs/.glo_dig_in_C5_CS1[6] <-> Connection Info Data/TwinSafeGroup_ES.Box 103 (EP1908) C5_CS1 - Module 1 (FSOE)_40 Info Data/Input Safe Data InputChannel6
//     RulliCentroTagliTask Inputs/.glo_dig_in_C5_CS1[7] <-> Connection Info Data/TwinSafeGroup_ES.Box 103 (EP1908) C5_CS1 - Module 1 (FSOE)_40 Info Data/Input Safe Data InputChannel7
//     RulliCentroTagliTask Inputs/.glo_dig_in_C5_CS1[8] <-> Connection Info Data/TwinSafeGroup_ES.Box 103 (EP1908) C5_CS1 - Module 1 (FSOE)_40 Info Data/Input Safe Data InputChannel8
//     RulliCentroTagliTask Inputs/.glo_dig_in_C3_CS1[{1..8}] <-> Connection Info Data/TwinSafeGroup_ES.Box 118 (EP1908) C3CS1 - Module 1 (FSOE)_39 Info Data/Input Safe Data InputChannel{1..8}  (8 links)
//     RulliCentroTagliTask Outputs/.TS_R1P1_Reset_Eme <-> StandardOutputs/TwinSafeGroup_ES.fromTC_R1P1_RestartE_Stop_RCS_41
//     RulliCentroTagliTask Outputs/.TS_R1P1_Reset_Eme_2 <-> StandardOutputs/TwinSafeGroup_ES.fromTC_R1P1_RestartE_Stop_RCS2_42
//   Galimberti/Galimberti Instance <-> Device 1 (EtherCAT)/Term 1 (EK1200) H-Q3/Term 5 (EK1110)
//     RulliCentroTagliTask Inputs/.glo_State_HQ3[4] <-> InfoData/State
//   Galimberti/Galimberti Instance <-> Device 1 (EtherCAT)/Term 39 (EK1100)/Term 40 (EL1008)
//     RulliCentroTagliTask Inputs/.glo_dig_in_Term_40[{1..8}] <-> Channel {1..8}/Input  (8 links)
//   Galimberti/Galimberti Instance <-> Device 1 (EtherCAT)/Term 39 (EK1100)/Term 46 (EK1122)/Box 47 (EP1008-0022) C1_CD4
//     RulliCentroTagliTask Inputs/.glo_State_C1CD4[1] <-> InfoData/State
//     RulliCentroTagliTask Inputs/.glo_WcState_C1CD4[1] <-> WcState/WcState
//     RulliCentroTagliTask Inputs/.glo_dig_in_C1CD4[{1..8}] <-> Channel {1..8}/Input  (8 links)
//   Galimberti/Galimberti Instance <-> Device 1 (EtherCAT)/Term 39 (EK1100)/Term 46 (EK1122)/Box 48 (EP6224-2022) C1_CO2
//     RulliCentroTagliTask Outputs/.glo_dig_out_C1CO2[1] <-> Module 3 (IO-Link Slave)/IO-Link Port1/Port1: process data
//     RulliCentroTagliTask Outputs/.glo_dig_out_C1CO2[2] <-> Module 4 (IO-Link Slave)/IO-Link Port2/Port2: process data
//   Galimberti/Galimberti Instance <-> Device 1 (EtherCAT)/Term 39 (EK1100)/Term 46 (EK1122)/Box 49 (EP1008-0022) C1_CD3
//     RulliCentroTagliTask Inputs/.glo_dig_in_C1CD3[{1..8}] <-> Channel {1..8}/Input  (8 links)
//   Galimberti/Galimberti Instance <-> Device 1 (EtherCAT)/Term 39 (EK1100)/Term 46 (EK1122)/Box 50 (EP6224-2022) C1_CO1
//     RulliCentroTagliTask Outputs/.glo_dig_out_C1CO1[{1..4}] <-> Module {3..6} (IO-Link Slave)/IO-Link Port{1..4}/Port{1..4}: process data  (4 links)
//   Galimberti/Galimberti Instance <-> Device 1 (EtherCAT)/Term 39 (EK1100)/Term 46 (EK1122)/Box 51 (EP1008-0022) C1_CD2
//     RulliCentroTagliTask Inputs/.glo_dig_in_C1CD2[{1..8}] <-> Channel {1..8}/Input  (8 links)
//   Galimberti/Galimberti Instance <-> Device 1 (EtherCAT)/Term 39 (EK1100)/Term 46 (EK1122)/Box 52 (EP1008-0022) C1_CD1
//     RulliCentroTagliTask Inputs/.glo_dig_in_C1CD1[{1..8}] <-> Channel {1..8}/Input  (8 links)
//   Galimberti/Galimberti Instance <-> Device 1 (EtherCAT)/Term 39 (EK1100)/Term 46 (EK1122)/Box 53 (EP1008-0022) C2_CD4
//     RulliCentroTagliTask Inputs/.glo_State_C2CD4[1] <-> InfoData/State
//     RulliCentroTagliTask Inputs/.glo_WcState_C2CD4[1] <-> WcState/WcState
//     RulliCentroTagliTask Inputs/.glo_dig_in_C2CD4[{1..8}] <-> Channel {1..8}/Input  (8 links)
//   Galimberti/Galimberti Instance <-> Device 1 (EtherCAT)/Term 39 (EK1100)/Term 46 (EK1122)/Box 54 (EP6228-0022) C2_CO1
//     RulliCentroTagliTask Inputs/.glo_dig_in_R1P5[1] <-> Module 9 (IO-Link Slave) - R1P5/IO-Link Port7_in/Switchstate Pin 1 (Bit0.0)
//     RulliCentroTagliTask Inputs/.glo_dig_in_R1P5[2] <-> Module 9 (IO-Link Slave) - R1P5/IO-Link Port7_in/Switchstate Pin 2 (Bit0.1)
//     RulliCentroTagliTask Inputs/.glo_dig_in_R1P5[3] <-> Module 9 (IO-Link Slave) - R1P5/IO-Link Port7_in/Switchstate Pin 3 (Bit0.2)
//     RulliCentroTagliTask Inputs/.glo_dig_in_R1P5[4] <-> Module 9 (IO-Link Slave) - R1P5/IO-Link Port7_in/Switchstate Pin 4 (Bit0.3)
//     RulliCentroTagliTask Inputs/.glo_dig_in_R1P5[5] <-> Module 9 (IO-Link Slave) - R1P5/IO-Link Port7_in/Switchstate Pin 5 (Bit0.4)
//     RulliCentroTagliTask Inputs/.glo_dig_in_R1P5[6] <-> Module 9 (IO-Link Slave) - R1P5/IO-Link Port7_in/Switchstate Pin 6 (Bit0.5)
//     RulliCentroTagliTask Inputs/.glo_dig_in_R1P5[7] <-> Module 9 (IO-Link Slave) - R1P5/IO-Link Port7_in/Switchstate Pin 7 (Bit0.6)
//     RulliCentroTagliTask Inputs/.glo_dig_in_R1P5[8] <-> Module 9 (IO-Link Slave) - R1P5/IO-Link Port7_in/Switchstate Pin 8 (Bit0.7)
//     RulliCentroTagliTask Inputs/.glo_dig_in_R1P6[1] <-> Module 10 (IO-Link Slave) - R1P6/IO-Link Port8_in/Switchstate Pin 1 (Bit0.0)
//     RulliCentroTagliTask Inputs/.glo_dig_in_R1P6[2] <-> Module 10 (IO-Link Slave) - R1P6/IO-Link Port8_in/Switchstate Pin 2 (Bit0.1)
//     RulliCentroTagliTask Inputs/.glo_dig_in_R1P6[3] <-> Module 10 (IO-Link Slave) - R1P6/IO-Link Port8_in/Switchstate Pin 3 (Bit0.2)
//     RulliCentroTagliTask Inputs/.glo_dig_in_R1P6[4] <-> Module 10 (IO-Link Slave) - R1P6/IO-Link Port8_in/Switchstate Pin 4 (Bit0.3)
//     RulliCentroTagliTask Inputs/.glo_dig_in_R1P6[5] <-> Module 10 (IO-Link Slave) - R1P6/IO-Link Port8_in/Switchstate Pin 5 (Bit0.4)
//     RulliCentroTagliTask Inputs/.glo_dig_in_R1P6[6] <-> Module 10 (IO-Link Slave) - R1P6/IO-Link Port8_in/Switchstate Pin 6 (Bit0.5)
//     RulliCentroTagliTask Inputs/.glo_dig_in_R1P6[7] <-> Module 10 (IO-Link Slave) - R1P6/IO-Link Port8_in/Switchstate Pin 7 (Bit0.6)
//     RulliCentroTagliTask Inputs/.glo_dig_in_R1P6[8] <-> Module 10 (IO-Link Slave) - R1P6/IO-Link Port8_in/Switchstate Pin 8 (Bit0.7)
//     RulliCentroTagliTask Outputs/.glo_dig_out_C2CO1[1] <-> Module 4 (IO-Link Slave)/IO-Link Port2/Port2: process data
//     RulliCentroTagliTask Outputs/.glo_dig_out_C2CO1[2] <-> Module 5 (IO-Link Slave)/IO-Link Port3/Port3: process data
//     RulliCentroTagliTask Outputs/.glo_dig_out_C2CO1[3] <-> Module 6 (IO-Link Slave)/IO-Link Port4/Port4: process data
//   Galimberti/Galimberti Instance <-> Device 1 (EtherCAT)/Term 39 (EK1100)/Term 46 (EK1122)/Box 55 (EP1008-0022) C2_CD3
//     RulliCentroTagliTask Inputs/.glo_dig_in_C2CD3[{1..8}] <-> Channel {1..8}/Input  (8 links)
//   Galimberti/Galimberti Instance <-> Device 1 (EtherCAT)/Term 39 (EK1100)/Term 46 (EK1122)/Box 56 (EP1008-0022) C2_CD2
//     RulliCentroTagliTask Inputs/.glo_dig_in_C2CD2[{1..8}] <-> Channel {1..8}/Input  (8 links)
//   Galimberti/Galimberti Instance <-> Device 1 (EtherCAT)/Term 39 (EK1100)/Term 46 (EK1122)/Box 57 (EP1008-0022) C2_CD1
//     RulliCentroTagliTask Inputs/.glo_dig_in_C2CD1[{1..8}] <-> Channel {1..8}/Input  (8 links)
//   Galimberti/Galimberti Instance <-> Device 1 (EtherCAT)/Term 39 (EK1100)/Term 46 (EK1122)/Box 58 (EP6228-0022) C2_CO2
//     RulliCentroTagliTask Inputs/.glo_IOLState_C2CO2[{1..8}] <-> Module 2 (DeviceState Inputs)/DeviceState Inputs/State Ch{1..8}  (8 links)
//     RulliCentroTagliTask Inputs/.glo_dig_in_C1P1[{1..8}] <-> Module 4 (IO-Link Slave) C1P1/IO-Link Port2_in/Switchstate Pin {1..8} (Bit0.{0..7})  (8 links)
//     RulliCentroTagliTask Inputs/.glo_dig_in_R1P1[1] <-> Module 6 (IO-Link Slave) R1P1/IO-Link Port4_in/Switchstate Pin 1 (Bit0.0)
//     RulliCentroTagliTask Inputs/.glo_dig_in_R1P1[2] <-> Module 6 (IO-Link Slave) R1P1/IO-Link Port4_in/Switchstate Pin 2 (Bit0.1)
//     RulliCentroTagliTask Inputs/.glo_dig_in_R1P1[3] <-> Module 6 (IO-Link Slave) R1P1/IO-Link Port4_in/Switchstate Pin 3 (Bit0.2)
//     RulliCentroTagliTask Inputs/.glo_dig_in_R1P1[4] <-> Module 6 (IO-Link Slave) R1P1/IO-Link Port4_in/Switchstate Pin 4 (Bit0.3)
//     RulliCentroTagliTask Inputs/.glo_dig_in_R1P1[5] <-> Module 6 (IO-Link Slave) R1P1/IO-Link Port4_in/Switchstate Pin 5 (Bit0.4)
//     RulliCentroTagliTask Inputs/.glo_dig_in_R1P1[6] <-> Module 6 (IO-Link Slave) R1P1/IO-Link Port4_in/Switchstate Pin 6 (Bit0.5)
//     RulliCentroTagliTask Inputs/.glo_dig_in_R1P1[7] <-> Module 6 (IO-Link Slave) R1P1/IO-Link Port4_in/Switchstate Pin 7 (Bit0.6)
//     RulliCentroTagliTask Inputs/.glo_dig_in_R1P1[8] <-> Module 6 (IO-Link Slave) R1P1/IO-Link Port4_in/Switchstate Pin 8 (Bit0.7)
//     RulliCentroTagliTask Inputs/.glo_dig_in_R1P1[9] <-> Module 6 (IO-Link Slave) R1P1/IO-Link Port4_in/Switchstate Pin 9 (Bit1.0)
//     RulliCentroTagliTask Inputs/.glo_dig_in_R1P2[1] <-> Module 7 (IO-Link Slave) R1P2/IO-Link Port5_in/Switchstate Pin 1 (Bit0.0)
//     RulliCentroTagliTask Inputs/.glo_dig_in_R1P2[2] <-> Module 7 (IO-Link Slave) R1P2/IO-Link Port5_in/Switchstate Pin 2 (Bit0.1)
//     RulliCentroTagliTask Inputs/.glo_dig_in_R1P2[3] <-> Module 7 (IO-Link Slave) R1P2/IO-Link Port5_in/Switchstate Pin 3 (Bit0.2)
//     RulliCentroTagliTask Inputs/.glo_dig_in_R1P2[4] <-> Module 7 (IO-Link Slave) R1P2/IO-Link Port5_in/Switchstate Pin 4 (Bit0.3)
//     RulliCentroTagliTask Inputs/.glo_dig_in_R1P2[5] <-> Module 7 (IO-Link Slave) R1P2/IO-Link Port5_in/Switchstate Pin 5 (Bit0.4)
//     RulliCentroTagliTask Inputs/.glo_dig_in_R1P2[6] <-> Module 7 (IO-Link Slave) R1P2/IO-Link Port5_in/Switchstate Pin 6 (Bit0.5)
//     RulliCentroTagliTask Inputs/.glo_dig_in_R1P2[7] <-> Module 7 (IO-Link Slave) R1P2/IO-Link Port5_in/Switchstate Pin 7 (Bit0.6)
//     RulliCentroTagliTask Inputs/.glo_dig_in_R1P2[8] <-> Module 7 (IO-Link Slave) R1P2/IO-Link Port5_in/Switchstate Pin 8 (Bit0.7)
//     RulliCentroTagliTask Inputs/.glo_dig_in_R1P3[1] <-> Module 8 (IO-Link Slave) R1P3/IO-Link Port6_in/Switchstate Pin 1 (Bit0.0)
//     RulliCentroTagliTask Inputs/.glo_dig_in_R1P3[2] <-> Module 8 (IO-Link Slave) R1P3/IO-Link Port6_in/Switchstate Pin 2 (Bit0.1)
//     RulliCentroTagliTask Inputs/.glo_dig_in_R1P3[3] <-> Module 8 (IO-Link Slave) R1P3/IO-Link Port6_in/Switchstate Pin 3 (Bit0.2)
//     RulliCentroTagliTask Inputs/.glo_dig_in_R1P3[4] <-> Module 8 (IO-Link Slave) R1P3/IO-Link Port6_in/Switchstate Pin 4 (Bit0.3)
//     RulliCentroTagliTask Inputs/.glo_dig_in_R1P3[5] <-> Module 8 (IO-Link Slave) R1P3/IO-Link Port6_in/Switchstate Pin 5 (Bit0.4)
//     RulliCentroTagliTask Inputs/.glo_dig_in_R1P3[6] <-> Module 8 (IO-Link Slave) R1P3/IO-Link Port6_in/Switchstate Pin 6 (Bit0.5)
//     RulliCentroTagliTask Inputs/.glo_dig_in_R1P3[7] <-> Module 8 (IO-Link Slave) R1P3/IO-Link Port6_in/Switchstate Pin 7 (Bit0.6)
//     RulliCentroTagliTask Inputs/.glo_dig_in_R1P3[8] <-> Module 8 (IO-Link Slave) R1P3/IO-Link Port6_in/Switchstate Pin 8 (Bit0.7)
//     RulliCentroTagliTask Inputs/.glo_dig_in_R1P4[1] <-> Module 9 (IO-Link Slave) R1P4/IO-Link Port7_in/Switchstate Pin 1 (Bit0.0)
//     RulliCentroTagliTask Inputs/.glo_dig_in_R1P4[2] <-> Module 9 (IO-Link Slave) R1P4/IO-Link Port7_in/Switchstate Pin 2 (Bit0.1)
//     RulliCentroTagliTask Inputs/.glo_dig_in_R1P4[3] <-> Module 9 (IO-Link Slave) R1P4/IO-Link Port7_in/Switchstate Pin 3 (Bit0.2)
//     RulliCentroTagliTask Inputs/.glo_dig_in_R1P4[4] <-> Module 9 (IO-Link Slave) R1P4/IO-Link Port7_in/Switchstate Pin 4 (Bit0.3)
//     RulliCentroTagliTask Inputs/.glo_dig_in_R1P4[5] <-> Module 9 (IO-Link Slave) R1P4/IO-Link Port7_in/Switchstate Pin 5 (Bit0.4)
//     RulliCentroTagliTask Inputs/.glo_dig_in_R1P4[6] <-> Module 9 (IO-Link Slave) R1P4/IO-Link Port7_in/Switchstate Pin 6 (Bit0.5)
//     RulliCentroTagliTask Inputs/.glo_dig_in_R1P4[7] <-> Module 9 (IO-Link Slave) R1P4/IO-Link Port7_in/Switchstate Pin 7 (Bit0.6)
//     RulliCentroTagliTask Inputs/.glo_dig_in_R1P4[8] <-> Module 9 (IO-Link Slave) R1P4/IO-Link Port7_in/Switchstate Pin 8 (Bit0.7)
//     RulliCentroTagliTask Outputs/.RCT_Semaforo.analog{0..5} <-> Module 10 (IO-Link Slave)/IO-Link Port8/Port8: process data[{0..5}]  (6 links)
//     RulliCentroTagliTask Outputs/.glo_dig_out_C1P1[{8..14}] <-> Module 4 (IO-Link Slave) C1P1/IO-Link Port2_out/Switchstate Pin {9..15} (Bit1.{0..6})  (7 links)
//     RulliCentroTagliTask Outputs/.glo_dig_out_R1P1[{10..16}] <-> Module 6 (IO-Link Slave) R1P1/IO-Link Port4_out/Switchstate Pin {10..16} (Bit1.{1..7})  (7 links)
//   Galimberti/Galimberti Instance <-> Device 1 (EtherCAT)/Term 39 (EK1100)/Term 61 (EK1122)/Box 100 (S100) R3
//     RulliCentroTagliTask Inputs/RULLI_CENTRO_TAGLI.R3_Inverter_Act_Alarm <-> Transmit PDO Mapping Parameter 3/subIndex 3
//     RulliCentroTagliTask Outputs/RULLI_CENTRO_TAGLI.R3_Inverter_Inverter_Cmd <-> Receive PDO Mapping Parameter 3/subIndex 2
//     RulliCentroTagliTask Outputs/RULLI_CENTRO_TAGLI.R3_Inverter_Speed_Override <-> Receive PDO Mapping Parameter 3/subIndex 1
//   Galimberti/Galimberti Instance <-> Device 1 (EtherCAT)/Term 39 (EK1100)/Term 61 (EK1122)/Box 101 (EP6228-0022) C5_CO1
//     RulliCentroTagliTask Outputs/.glo_dig_out_C5CO1[1] <-> Module 3 (IO-Link Slave)/IO-Link Port1/Port1: process data
//     RulliCentroTagliTask Outputs/.glo_dig_out_C5CO1[2] <-> Module 4 (IO-Link Slave)/IO-Link Port2/Port2: process data
//     RulliCentroTagliTask Outputs/.glo_dig_out_C5CO1[3] <-> Module 5 (IO-Link Slave)/IO-Link Port3/Port3: process data
//     RulliCentroTagliTask Outputs/.glo_dig_out_C5CO1[4] <-> Module 7 (IO-Link Slave)/IO-Link Port5/Port5: process data
//     RulliCentroTagliTask Outputs/.glo_dig_out_C5CO1[5] <-> Module 8 (IO-Link Slave)/IO-Link Port6/Port6: process data
//     RulliCentroTagliTask Outputs/.glo_dig_out_C5CO1[6] <-> Module 9 (IO-Link Slave)/IO-Link Port7/Port7: process data
//   Galimberti/Galimberti Instance <-> Device 1 (EtherCAT)/Term 39 (EK1100)/Term 61 (EK1122)/Box 102 (EP1008-0022) C5_CD1
//     RulliCentroTagliTask Inputs/.glo_dig_in_C5CD1[{1..8}] <-> Channel {1..8}/Input  (8 links)
//   Galimberti/Galimberti Instance <-> Device 1 (EtherCAT)/Term 39 (EK1100)/Term 61 (EK1122)/Box 104 (EP6228-0022) C5_CO2
//     RulliCentroTagliTask Inputs/.glo_dig_in_C5CO2[1] <-> Module 5 (IO-Link Slave)/IO-Link Port3/Port3: process data
//     RulliCentroTagliTask Inputs/.glo_dig_in_C5CO2[2] <-> Module 6 (IO-Link Slave)/IO-Link Port4/Port4: process data
//     RulliCentroTagliTask Inputs/.glo_dig_in_R3P1[1] <-> Module 7 (IO-Link Slave)/IO-Link Port5_in/Switchstate Pin 1 (Bit0.0)
//     RulliCentroTagliTask Inputs/.glo_dig_in_R3P1[2] <-> Module 7 (IO-Link Slave)/IO-Link Port5_in/Switchstate Pin 2 (Bit0.1)
//     RulliCentroTagliTask Inputs/.glo_dig_in_R3P1[3] <-> Module 7 (IO-Link Slave)/IO-Link Port5_in/Switchstate Pin 3 (Bit0.2)
//     RulliCentroTagliTask Inputs/.glo_dig_in_R3P1[4] <-> Module 7 (IO-Link Slave)/IO-Link Port5_in/Switchstate Pin 4 (Bit0.3)
//     RulliCentroTagliTask Inputs/.glo_dig_in_R3P1[5] <-> Module 7 (IO-Link Slave)/IO-Link Port5_in/Switchstate Pin 5 (Bit0.4)
//     RulliCentroTagliTask Inputs/.glo_dig_in_R3P1[6] <-> Module 7 (IO-Link Slave)/IO-Link Port5_in/Switchstate Pin 6 (Bit0.5)
//     RulliCentroTagliTask Inputs/.glo_dig_in_R3P1[7] <-> Module 7 (IO-Link Slave)/IO-Link Port5_in/Switchstate Pin 7 (Bit0.6)
//     RulliCentroTagliTask Inputs/.glo_dig_in_R3P1[8] <-> Module 7 (IO-Link Slave)/IO-Link Port5_in/Switchstate Pin 8 (Bit0.7)
//     RulliCentroTagliTask Inputs/.glo_dig_in_R3P2[1] <-> Module 8 (IO-Link Slave)/IO-Link Port6_in/Switchstate Pin 1 (Bit0.0)
//     RulliCentroTagliTask Inputs/.glo_dig_in_R3P2[2] <-> Module 8 (IO-Link Slave)/IO-Link Port6_in/Switchstate Pin 2 (Bit0.1)
//     RulliCentroTagliTask Inputs/.glo_dig_in_R3P2[3] <-> Module 8 (IO-Link Slave)/IO-Link Port6_in/Switchstate Pin 3 (Bit0.2)
//     RulliCentroTagliTask Inputs/.glo_dig_in_R3P2[4] <-> Module 8 (IO-Link Slave)/IO-Link Port6_in/Switchstate Pin 4 (Bit0.3)
//     RulliCentroTagliTask Inputs/.glo_dig_in_R3P2[5] <-> Module 8 (IO-Link Slave)/IO-Link Port6_in/Switchstate Pin 5 (Bit0.4)
//     RulliCentroTagliTask Inputs/.glo_dig_in_R3P2[6] <-> Module 8 (IO-Link Slave)/IO-Link Port6_in/Switchstate Pin 6 (Bit0.5)
//     RulliCentroTagliTask Inputs/.glo_dig_in_R3P2[7] <-> Module 8 (IO-Link Slave)/IO-Link Port6_in/Switchstate Pin 7 (Bit0.6)
//     RulliCentroTagliTask Inputs/.glo_dig_in_R3P2[8] <-> Module 8 (IO-Link Slave)/IO-Link Port6_in/Switchstate Pin 8 (Bit0.7)
//     RulliCentroTagliTask Inputs/.glo_dig_in_R3P3[1] <-> Module 9 (IO-Link Slave)/IO-Link Port7_in/Switchstate Pin 1 (Bit0.0)
//     RulliCentroTagliTask Inputs/.glo_dig_in_R3P3[2] <-> Module 9 (IO-Link Slave)/IO-Link Port7_in/Switchstate Pin 2 (Bit0.1)
//     RulliCentroTagliTask Inputs/.glo_dig_in_R3P3[3] <-> Module 9 (IO-Link Slave)/IO-Link Port7_in/Switchstate Pin 3 (Bit0.2)
//     RulliCentroTagliTask Inputs/.glo_dig_in_R3P3[4] <-> Module 9 (IO-Link Slave)/IO-Link Port7_in/Switchstate Pin 4 (Bit0.3)
//     RulliCentroTagliTask Inputs/.glo_dig_in_R3P3[5] <-> Module 9 (IO-Link Slave)/IO-Link Port7_in/Switchstate Pin 5 (Bit0.4)
//     RulliCentroTagliTask Inputs/.glo_dig_in_R3P3[6] <-> Module 9 (IO-Link Slave)/IO-Link Port7_in/Switchstate Pin 6 (Bit0.5)
//     RulliCentroTagliTask Inputs/.glo_dig_in_R3P3[7] <-> Module 9 (IO-Link Slave)/IO-Link Port7_in/Switchstate Pin 7 (Bit0.6)
//     RulliCentroTagliTask Inputs/.glo_dig_in_R3P3[8] <-> Module 9 (IO-Link Slave)/IO-Link Port7_in/Switchstate Pin 8 (Bit0.7)
//     RulliCentroTagliTask Inputs/.glo_dig_in_R3P4[10] <-> Module 10 (IO-Link Slave)/IO-Link Port8_in/Switchstate Pin 10 (Bit1.1)
//     RulliCentroTagliTask Inputs/.glo_dig_in_R3P4[11] <-> Module 10 (IO-Link Slave)/IO-Link Port8_in/Switchstate Pin 11 (Bit1.2)
//     RulliCentroTagliTask Inputs/.glo_dig_in_R3P4[12] <-> Module 10 (IO-Link Slave)/IO-Link Port8_in/Switchstate Pin 12 (Bit1.3)
//     RulliCentroTagliTask Inputs/.glo_dig_in_R3P4[13] <-> Module 10 (IO-Link Slave)/IO-Link Port8_in/Switchstate Pin 13 (Bit1.4)
//     RulliCentroTagliTask Inputs/.glo_dig_in_R3P4[14] <-> Module 10 (IO-Link Slave)/IO-Link Port8_in/Switchstate Pin 14 (Bit1.5)
//     RulliCentroTagliTask Inputs/.glo_dig_in_R3P4[15] <-> Module 10 (IO-Link Slave)/IO-Link Port8_in/Switchstate Pin 15 (Bit1.6)
//     RulliCentroTagliTask Inputs/.glo_dig_in_R3P4[16] <-> Module 10 (IO-Link Slave)/IO-Link Port8_in/Switchstate Pin 16 (Bit1.7)
//     RulliCentroTagliTask Inputs/.glo_dig_in_R3P4[1] <-> Module 10 (IO-Link Slave)/IO-Link Port8_in/Switchstate Pin 1 (Bit0.0)
//     RulliCentroTagliTask Inputs/.glo_dig_in_R3P4[2] <-> Module 10 (IO-Link Slave)/IO-Link Port8_in/Switchstate Pin 2 (Bit0.1)
//     RulliCentroTagliTask Inputs/.glo_dig_in_R3P4[3] <-> Module 10 (IO-Link Slave)/IO-Link Port8_in/Switchstate Pin 3 (Bit0.2)
//     RulliCentroTagliTask Inputs/.glo_dig_in_R3P4[4] <-> Module 10 (IO-Link Slave)/IO-Link Port8_in/Switchstate Pin 4 (Bit0.3)
//     RulliCentroTagliTask Inputs/.glo_dig_in_R3P4[5] <-> Module 10 (IO-Link Slave)/IO-Link Port8_in/Switchstate Pin 5 (Bit0.4)
//     RulliCentroTagliTask Inputs/.glo_dig_in_R3P4[6] <-> Module 10 (IO-Link Slave)/IO-Link Port8_in/Switchstate Pin 6 (Bit0.5)
//     RulliCentroTagliTask Inputs/.glo_dig_in_R3P4[7] <-> Module 10 (IO-Link Slave)/IO-Link Port8_in/Switchstate Pin 7 (Bit0.6)
//     RulliCentroTagliTask Inputs/.glo_dig_in_R3P4[8] <-> Module 10 (IO-Link Slave)/IO-Link Port8_in/Switchstate Pin 8 (Bit0.7)
//     RulliCentroTagliTask Inputs/.glo_dig_in_R3P4[9] <-> Module 10 (IO-Link Slave)/IO-Link Port8_in/Switchstate Pin 9 (Bit1.0)
//     RulliCentroTagliTask Outputs/.glo_dig_out_C5CO2[1] <-> Module 3 (IO-Link Slave)/IO-Link Port1/Port1: process data
//     RulliCentroTagliTask Outputs/.glo_dig_out_C5CO2[2] <-> Module 4 (IO-Link Slave)/IO-Link Port2/Port2: process data
//     RulliCentroTagliTask Outputs/.glo_dig_out_R3P4[10] <-> Module 10 (IO-Link Slave)/IO-Link Port8_out/Switchstate Pin 10 (Bit1.1)
//     RulliCentroTagliTask Outputs/.glo_dig_out_R3P4[11] <-> Module 10 (IO-Link Slave)/IO-Link Port8_out/Switchstate Pin 11 (Bit1.2)
//     RulliCentroTagliTask Outputs/.glo_dig_out_R3P4[12] <-> Module 10 (IO-Link Slave)/IO-Link Port8_out/Switchstate Pin 12 (Bit1.3)
//     RulliCentroTagliTask Outputs/.glo_dig_out_R3P4[13] <-> Module 10 (IO-Link Slave)/IO-Link Port8_out/Switchstate Pin 13 (Bit1.4)
//     RulliCentroTagliTask Outputs/.glo_dig_out_R3P4[14] <-> Module 10 (IO-Link Slave)/IO-Link Port8_out/Switchstate Pin 14 (Bit1.5)
//     RulliCentroTagliTask Outputs/.glo_dig_out_R3P4[15] <-> Module 10 (IO-Link Slave)/IO-Link Port8_out/Switchstate Pin 15 (Bit1.6)
//     RulliCentroTagliTask Outputs/.glo_dig_out_R3P4[16] <-> Module 10 (IO-Link Slave)/IO-Link Port8_out/Switchstate Pin 16 (Bit1.7)
//     RulliCentroTagliTask Outputs/.glo_dig_out_R3P4[1] <-> Module 10 (IO-Link Slave)/IO-Link Port8_out/Switchstate Pin 1 (Bit0.0)
//     RulliCentroTagliTask Outputs/.glo_dig_out_R3P4[2] <-> Module 10 (IO-Link Slave)/IO-Link Port8_out/Switchstate Pin 2 (Bit0.1)
//     RulliCentroTagliTask Outputs/.glo_dig_out_R3P4[3] <-> Module 10 (IO-Link Slave)/IO-Link Port8_out/Switchstate Pin 3 (Bit0.2)
//     RulliCentroTagliTask Outputs/.glo_dig_out_R3P4[4] <-> Module 10 (IO-Link Slave)/IO-Link Port8_out/Switchstate Pin 4 (Bit0.3)
//     RulliCentroTagliTask Outputs/.glo_dig_out_R3P4[5] <-> Module 10 (IO-Link Slave)/IO-Link Port8_out/Switchstate Pin 5 (Bit0.4)
//     RulliCentroTagliTask Outputs/.glo_dig_out_R3P4[6] <-> Module 10 (IO-Link Slave)/IO-Link Port8_out/Switchstate Pin 6 (Bit0.5)
//     RulliCentroTagliTask Outputs/.glo_dig_out_R3P4[7] <-> Module 10 (IO-Link Slave)/IO-Link Port8_out/Switchstate Pin 7 (Bit0.6)
//     RulliCentroTagliTask Outputs/.glo_dig_out_R3P4[8] <-> Module 10 (IO-Link Slave)/IO-Link Port8_out/Switchstate Pin 8 (Bit0.7)
//     RulliCentroTagliTask Outputs/.glo_dig_out_R3P4[9] <-> Module 10 (IO-Link Slave)/IO-Link Port8_out/Switchstate Pin 9 (Bit1.0)
//   Galimberti/Galimberti Instance <-> Device 1 (EtherCAT)/Term 39 (EK1100)/Term 61 (EK1122)/Box 105 (EP1008-0022) C5_CD2
//     RulliCentroTagliTask Inputs/.glo_dig_in_C5CD2[{1..8}] <-> Channel {1..8}/Input  (8 links)
//   Galimberti/Galimberti Instance <-> Device 1 (EtherCAT)/Term 39 (EK1100)/Term 61 (EK1122)/Box 106 (EP1008-0022) C5_CD3
//     RulliCentroTagliTask Inputs/.glo_dig_in_C5CD3[{1..8}] <-> Channel {1..8}/Input  (8 links)
//   Galimberti/Galimberti Instance <-> Device 1 (EtherCAT)/Term 39 (EK1100)/Term 61 (EK1122)/Box 115 (EP1008-0022) C3CD1
//     RulliCentroTagliTask Inputs/.glo_dig_in_C3CD1[{1..8}] <-> Channel {1..8}/Input  (8 links)
//   Galimberti/Galimberti Instance <-> Device 1 (EtherCAT)/Term 39 (EK1100)/Term 61 (EK1122)/Box 116 (EP6228-0022) C3CO1
//     RulliCentroTagliTask Inputs/.glo_dig_in_C3CO1[1] <-> Module 10 (IO-Link Slave)/IO-Link Port8/Port8: process data
//     RulliCentroTagliTask Inputs/.glo_dig_in_C4P1[10] <-> Module 8 (IO-Link Slave)/IO-Link Port6_in/Switchstate Pin 10 (Bit1.1)
//     RulliCentroTagliTask Inputs/.glo_dig_in_C4P1[11] <-> Module 8 (IO-Link Slave)/IO-Link Port6_in/Switchstate Pin 11 (Bit1.2)
//     RulliCentroTagliTask Inputs/.glo_dig_in_C4P1[12] <-> Module 8 (IO-Link Slave)/IO-Link Port6_in/Switchstate Pin 12 (Bit1.3)
//     RulliCentroTagliTask Inputs/.glo_dig_in_C4P1[13] <-> Module 8 (IO-Link Slave)/IO-Link Port6_in/Switchstate Pin 13 (Bit1.4)
//     RulliCentroTagliTask Inputs/.glo_dig_in_C4P1[14] <-> Module 8 (IO-Link Slave)/IO-Link Port6_in/Switchstate Pin 14 (Bit1.5)
//     RulliCentroTagliTask Inputs/.glo_dig_in_C4P1[15] <-> Module 8 (IO-Link Slave)/IO-Link Port6_in/Switchstate Pin 15 (Bit1.6)
//     RulliCentroTagliTask Inputs/.glo_dig_in_C4P1[16] <-> Module 8 (IO-Link Slave)/IO-Link Port6_in/Switchstate Pin 16 (Bit1.7)
//     RulliCentroTagliTask Inputs/.glo_dig_in_C4P1[1] <-> Module 8 (IO-Link Slave)/IO-Link Port6_in/Switchstate Pin 1 (Bit0.0)
//     RulliCentroTagliTask Inputs/.glo_dig_in_C4P1[2] <-> Module 8 (IO-Link Slave)/IO-Link Port6_in/Switchstate Pin 2 (Bit0.1)
//     RulliCentroTagliTask Inputs/.glo_dig_in_C4P1[3] <-> Module 8 (IO-Link Slave)/IO-Link Port6_in/Switchstate Pin 3 (Bit0.2)
//     RulliCentroTagliTask Inputs/.glo_dig_in_C4P1[4] <-> Module 8 (IO-Link Slave)/IO-Link Port6_in/Switchstate Pin 4 (Bit0.3)
//     RulliCentroTagliTask Inputs/.glo_dig_in_C4P1[5] <-> Module 8 (IO-Link Slave)/IO-Link Port6_in/Switchstate Pin 5 (Bit0.4)
//     RulliCentroTagliTask Inputs/.glo_dig_in_C4P1[6] <-> Module 8 (IO-Link Slave)/IO-Link Port6_in/Switchstate Pin 6 (Bit0.5)
//     RulliCentroTagliTask Inputs/.glo_dig_in_C4P1[7] <-> Module 8 (IO-Link Slave)/IO-Link Port6_in/Switchstate Pin 7 (Bit0.6)
//     RulliCentroTagliTask Inputs/.glo_dig_in_C4P1[8] <-> Module 8 (IO-Link Slave)/IO-Link Port6_in/Switchstate Pin 8 (Bit0.7)
//     RulliCentroTagliTask Inputs/.glo_dig_in_C4P1[9] <-> Module 8 (IO-Link Slave)/IO-Link Port6_in/Switchstate Pin 9 (Bit1.0)
//     RulliCentroTagliTask Inputs/.glo_dig_in_C4PO1[{1..8}] <-> Module 9 (IO-Link Slave)/IO-Link Port7_in/Switchstate Pin {1..8} (Bit0.{0..7})  (8 links)
//     RulliCentroTagliTask Outputs/.glo_dig_out_C3CO1[2] <-> Module 4 (IO-Link Slave)/IO-Link Port2/Port2: process data
//     RulliCentroTagliTask Outputs/.glo_dig_out_C3CO1[3] <-> Module 5 (IO-Link Slave)/IO-Link Port3/Port3: process data
//     RulliCentroTagliTask Outputs/.glo_dig_out_C4P1[10] <-> Module 8 (IO-Link Slave)/IO-Link Port6_out/Switchstate Pin 10 (Bit1.1)
//     RulliCentroTagliTask Outputs/.glo_dig_out_C4P1[11] <-> Module 8 (IO-Link Slave)/IO-Link Port6_out/Switchstate Pin 11 (Bit1.2)
//     RulliCentroTagliTask Outputs/.glo_dig_out_C4P1[12] <-> Module 8 (IO-Link Slave)/IO-Link Port6_out/Switchstate Pin 12 (Bit1.3)
//     RulliCentroTagliTask Outputs/.glo_dig_out_C4P1[13] <-> Module 8 (IO-Link Slave)/IO-Link Port6_out/Switchstate Pin 13 (Bit1.4)
//     RulliCentroTagliTask Outputs/.glo_dig_out_C4P1[14] <-> Module 8 (IO-Link Slave)/IO-Link Port6_out/Switchstate Pin 14 (Bit1.5)
//     RulliCentroTagliTask Outputs/.glo_dig_out_C4P1[15] <-> Module 8 (IO-Link Slave)/IO-Link Port6_out/Switchstate Pin 15 (Bit1.6)
//     RulliCentroTagliTask Outputs/.glo_dig_out_C4P1[16] <-> Module 8 (IO-Link Slave)/IO-Link Port6_out/Switchstate Pin 16 (Bit1.7)
//     RulliCentroTagliTask Outputs/.glo_dig_out_C4P1[1] <-> Module 8 (IO-Link Slave)/IO-Link Port6_out/Switchstate Pin 1 (Bit0.0)
//     RulliCentroTagliTask Outputs/.glo_dig_out_C4P1[2] <-> Module 8 (IO-Link Slave)/IO-Link Port6_out/Switchstate Pin 2 (Bit0.1)
//     RulliCentroTagliTask Outputs/.glo_dig_out_C4P1[3] <-> Module 8 (IO-Link Slave)/IO-Link Port6_out/Switchstate Pin 3 (Bit0.2)
//     RulliCentroTagliTask Outputs/.glo_dig_out_C4P1[4] <-> Module 8 (IO-Link Slave)/IO-Link Port6_out/Switchstate Pin 4 (Bit0.3)
//     RulliCentroTagliTask Outputs/.glo_dig_out_C4P1[5] <-> Module 8 (IO-Link Slave)/IO-Link Port6_out/Switchstate Pin 5 (Bit0.4)
//     RulliCentroTagliTask Outputs/.glo_dig_out_C4P1[6] <-> Module 8 (IO-Link Slave)/IO-Link Port6_out/Switchstate Pin 6 (Bit0.5)
//     RulliCentroTagliTask Outputs/.glo_dig_out_C4P1[7] <-> Module 8 (IO-Link Slave)/IO-Link Port6_out/Switchstate Pin 7 (Bit0.6)
//     RulliCentroTagliTask Outputs/.glo_dig_out_C4P1[8] <-> Module 8 (IO-Link Slave)/IO-Link Port6_out/Switchstate Pin 8 (Bit0.7)
//     RulliCentroTagliTask Outputs/.glo_dig_out_C4P1[9] <-> Module 8 (IO-Link Slave)/IO-Link Port6_out/Switchstate Pin 9 (Bit1.0)
//   Galimberti/Galimberti Instance <-> Device 1 (EtherCAT)/Term 39 (EK1100)/Term 61 (EK1122)/Box 117 (EP1008-0022) C3CD2
//     RulliCentroTagliTask Inputs/.glo_dig_in_C3CD2[{1..8}] <-> Channel {1..8}/Input  (8 links)
//   Galimberti/Galimberti Instance <-> Device 1 (EtherCAT)/Term 39 (EK1100)/Term 61 (EK1122)/Box 68 (S100) R1M2
//     RulliCentroTagliTask Inputs/RULLI_CENTRO_TAGLI.R1_Inverter_Act_Alarm <-> Transmit PDO Mapping Parameter 3/SubIndex 003
//     RulliCentroTagliTask Outputs/RULLI_CENTRO_TAGLI.R1_Inverter_Inverter_Cmd <-> Receive PDO Mapping Parameter 3/SubIndex 002
//     RulliCentroTagliTask Outputs/RULLI_CENTRO_TAGLI.R1_Inverter_Speed_Override <-> Receive PDO Mapping Parameter 3/SubIndex 001
//   Galimberti/Galimberti Instance <-> Device 1 (EtherCAT)/Term 39 (EK1100)/Term 61 (EK1122)/Box 99 (S100) R2
//     RulliCentroTagliTask Inputs/RULLI_CENTRO_TAGLI.R2_Inverter_Act_Alarm <-> Transmit PDO Mapping Parameter 3/subIndex 3
//     RulliCentroTagliTask Outputs/RULLI_CENTRO_TAGLI.R2_Inverter_Inverter_Cmd <-> Receive PDO Mapping Parameter 3/subIndex 2
//     RulliCentroTagliTask Outputs/RULLI_CENTRO_TAGLI.R2_Inverter_Speed_Override <-> Receive PDO Mapping Parameter 3/subIndex 1
//   Galimberti/Galimberti Instance <-> Device 1 (EtherCAT)/Term 6 (EK1100) H-Q1/Term 10 (EL2008)
//     PlcTask Outputs/.glo_dig_out_HQ1[{9..16}] <-> Channel {1..8}/Output  (8 links)
//     RulliCentroTagliTask Inputs/.glo_State_HQ1[4] <-> InfoData/State
//     RulliCentroTagliTask Inputs/.glo_WcState_HQ1[4] <-> WcState/WcState
//   Galimberti/Galimberti Instance <-> Device 1 (EtherCAT)/Term 6 (EK1100) H-Q1/Term 11 (EL3012)
//     PlcTask Inputs/.glo_analog_in_HQ1[1] <-> AI Standard Channel 1/Value
//     PlcTask Inputs/.glo_analog_in_HQ1[2] <-> AI Standard Channel 2/Value
//     RulliCentroTagliTask Inputs/.glo_State_HQ1[5] <-> InfoData/State
//     RulliCentroTagliTask Inputs/.glo_WcState_HQ1[5] <-> WcState/WcState
//   Galimberti/Galimberti Instance <-> Device 1 (EtherCAT)/Term 6 (EK1100) H-Q1/Term 12 (EL3012)
//     PlcTask Inputs/.glo_analog_in_HQ1[3] <-> AI Standard Channel 1/Value
//     PlcTask Inputs/.glo_analog_in_HQ1[4] <-> AI Standard Channel 2/Value
//     RulliCentroTagliTask Inputs/.glo_State_HQ1[6] <-> InfoData/State
//     RulliCentroTagliTask Inputs/.glo_WcState_HQ1[6] <-> WcState/WcState
//   Galimberti/Galimberti Instance <-> Device 1 (EtherCAT)/Term 6 (EK1100) H-Q1/Term 13 (EL2904)
//     RulliCentroTagliTask Inputs/.glo_State_HQ1[7] <-> InfoData/State
//     RulliCentroTagliTask Inputs/.glo_WcState_HQ1[7] <-> WcState/WcState
//   Galimberti/Galimberti Instance <-> Device 1 (EtherCAT)/Term 6 (EK1100) H-Q1/Term 14 (EL2904)
//     RulliCentroTagliTask Inputs/.glo_State_HQ1[8] <-> InfoData/State
//     RulliCentroTagliTask Inputs/.glo_WcState_HQ1[8] <-> WcState/WcState
//   Galimberti/Galimberti Instance <-> Device 1 (EtherCAT)/Term 6 (EK1100) H-Q1/Term 15 (EK1110)
//     RulliCentroTagliTask Inputs/.glo_State_HQ1[9] <-> InfoData/State
//   Galimberti/Galimberti Instance <-> Device 1 (EtherCAT)/Term 6 (EK1100) H-Q1/Term 35 (EL6695)
//     RulliCentroTagliTask Inputs/.RD_Aspirazione_RUN <-> IO Inputs/Var 17173
//     RulliCentroTagliTask Outputs/.WR_Req_Start_Aspirazione <-> IO Outputs/Var 17174
//   Galimberti/Galimberti Instance <-> Device 1 (EtherCAT)/Term 6 (EK1100) H-Q1/Term 7 (EL1008)
//     PlcTask Inputs/.glo_dig_in_HQ1[{1..8}] <-> Channel {1..8}/Input  (8 links)
//     RulliCentroTagliTask Inputs/.glo_State_HQ1[1] <-> InfoData/State
//     RulliCentroTagliTask Inputs/.glo_WcState_HQ1[1] <-> WcState/WcState
//   Galimberti/Galimberti Instance <-> Device 1 (EtherCAT)/Term 6 (EK1100) H-Q1/Term 8 (EL1008)
//     PlcTask Inputs/.glo_dig_in_HQ1[{9..16}] <-> Channel {1..8}/Input  (8 links)
//     RulliCentroTagliTask Inputs/.glo_State_HQ1[2] <-> InfoData/State
//     RulliCentroTagliTask Inputs/.glo_WcState_HQ1[2] <-> WcState/WcState
//   Galimberti/Galimberti Instance <-> Device 1 (EtherCAT)/Term 6 (EK1100) H-Q1/Term 9 (EL2008)
//     PlcTask Outputs/.glo_dig_out_HQ1[{1..8}] <-> Channel {1..8}/Output  (8 links)
//     RulliCentroTagliTask Inputs/.glo_State_HQ1[3] <-> InfoData/State
//     RulliCentroTagliTask Inputs/.glo_WcState_HQ1[3] <-> WcState/WcState
//   Galimberti/Galimberti Instance <-> NC-Task 1 SAF/Axes/C1M1
//     RulliCentroTagliTask Inputs/RULLI_CENTRO_TAGLI.Catenaria_C1_Solleva.NcToPlc <-> Outputs/ToPlc
//     RulliCentroTagliTask Inputs/RULLI_CENTRO_TAGLI.Catenaria_C1_Solleva_Status_Dword/CamDataQueued <-> Outputs/ToPlc/StateDWord/CamDataQueued
//     RulliCentroTagliTask Inputs/RULLI_CENTRO_TAGLI.Catenaria_C1_Solleva_Status_Dword/CamScalingPending <-> Outputs/ToPlc/StateDWord/CamScalingPending
//     RulliCentroTagliTask Inputs/RULLI_CENTRO_TAGLI.Catenaria_C1_Solleva_Status_Dword/CamTableQueued <-> Outputs/ToPlc/StateDWord/CamTableQueued
//     RulliCentroTagliTask Inputs/RULLI_CENTRO_TAGLI.Catenaria_C1_Solleva_Status_Dword/CmdBuffered <-> Outputs/ToPlc/StateDWord/CmdBuffered
//     RulliCentroTagliTask Inputs/RULLI_CENTRO_TAGLI.Catenaria_C1_Solleva_Status_Dword/Compensating <-> Outputs/ToPlc/StateDWord/Compensating
//     RulliCentroTagliTask Inputs/RULLI_CENTRO_TAGLI.Catenaria_C1_Solleva_Status_Dword/ConstantVelocity <-> Outputs/ToPlc/StateDWord/ConstantVelocity
//     RulliCentroTagliTask Inputs/RULLI_CENTRO_TAGLI.Catenaria_C1_Solleva_Status_Dword/ContinuousMotion <-> Outputs/ToPlc/StateDWord/ContinuousMotion
//     RulliCentroTagliTask Inputs/RULLI_CENTRO_TAGLI.Catenaria_C1_Solleva_Status_Dword/ControlLoopClosed <-> Outputs/ToPlc/StateDWord/ControlLoopClosed
//     RulliCentroTagliTask Inputs/RULLI_CENTRO_TAGLI.Catenaria_C1_Solleva_Status_Dword/DriveDeviceError <-> Outputs/ToPlc/StateDWord/DriveDeviceError
//     RulliCentroTagliTask Inputs/RULLI_CENTRO_TAGLI.Catenaria_C1_Solleva_Status_Dword/ErrorPropagationDelayed <-> Outputs/ToPlc/StateDWord/ErrorPropagationDelayed
//     RulliCentroTagliTask Inputs/RULLI_CENTRO_TAGLI.Catenaria_C1_Solleva_Status_Dword/ExtSetPointGenEnabled <-> Outputs/ToPlc/StateDWord/ExtSetPointGenEnabled
//     RulliCentroTagliTask Inputs/RULLI_CENTRO_TAGLI.Catenaria_C1_Solleva_Status_Dword/ExternalLatchValid <-> Outputs/ToPlc/StateDWord/ExternalLatchValid
//     RulliCentroTagliTask Inputs/RULLI_CENTRO_TAGLI.Catenaria_C1_Solleva_Status_Dword/HasBeenStopped <-> Outputs/ToPlc/StateDWord/HasBeenStopped
//     RulliCentroTagliTask Inputs/RULLI_CENTRO_TAGLI.Catenaria_C1_Solleva_Status_Dword/HasJob <-> Outputs/ToPlc/StateDWord/HasJob
//     RulliCentroTagliTask Inputs/RULLI_CENTRO_TAGLI.Catenaria_C1_Solleva_Status_Dword/Homed <-> Outputs/ToPlc/StateDWord/Homed
//     RulliCentroTagliTask Inputs/RULLI_CENTRO_TAGLI.Catenaria_C1_Solleva_Status_Dword/HomingBusy <-> Outputs/ToPlc/StateDWord/HomingBusy
//     RulliCentroTagliTask Inputs/RULLI_CENTRO_TAGLI.Catenaria_C1_Solleva_Status_Dword/InPositionArea <-> Outputs/ToPlc/StateDWord/InPositionArea
//     RulliCentroTagliTask Inputs/RULLI_CENTRO_TAGLI.Catenaria_C1_Solleva_Status_Dword/InTargetPosition <-> Outputs/ToPlc/StateDWord/InTargetPosition
//     RulliCentroTagliTask Inputs/RULLI_CENTRO_TAGLI.Catenaria_C1_Solleva_Status_Dword/IoDataInvalid <-> Outputs/ToPlc/StateDWord/IoDataInvalid
//     RulliCentroTagliTask Inputs/RULLI_CENTRO_TAGLI.Catenaria_C1_Solleva_Status_Dword/MotionCommandsLocked <-> Outputs/ToPlc/StateDWord/MotionCommandsLocked
//     RulliCentroTagliTask Inputs/RULLI_CENTRO_TAGLI.Catenaria_C1_Solleva_Status_Dword/NegativeDirection <-> Outputs/ToPlc/StateDWord/NegativeDirection
//     RulliCentroTagliTask Inputs/RULLI_CENTRO_TAGLI.Catenaria_C1_Solleva_Status_Dword/NewTargetPos <-> Outputs/ToPlc/StateDWord/NewTargetPos
//     RulliCentroTagliTask Inputs/RULLI_CENTRO_TAGLI.Catenaria_C1_Solleva_Status_Dword/NotMoving <-> Outputs/ToPlc/StateDWord/NotMoving
//     RulliCentroTagliTask Inputs/RULLI_CENTRO_TAGLI.Catenaria_C1_Solleva_Status_Dword/Operational <-> Outputs/ToPlc/StateDWord/Operational
//     RulliCentroTagliTask Inputs/RULLI_CENTRO_TAGLI.Catenaria_C1_Solleva_Status_Dword/PTPmode <-> Outputs/ToPlc/StateDWord/PTPmode
//     RulliCentroTagliTask Inputs/RULLI_CENTRO_TAGLI.Catenaria_C1_Solleva_Status_Dword/PhasingActive <-> Outputs/ToPlc/StateDWord/PhasingActive
//     RulliCentroTagliTask Inputs/RULLI_CENTRO_TAGLI.Catenaria_C1_Solleva_Status_Dword/PositiveDirection <-> Outputs/ToPlc/StateDWord/PositiveDirection
//     RulliCentroTagliTask Inputs/RULLI_CENTRO_TAGLI.Catenaria_C1_Solleva_Status_Dword/Protected_ <-> Outputs/ToPlc/StateDWord/Protected
//     RulliCentroTagliTask Inputs/RULLI_CENTRO_TAGLI.Catenaria_C1_Solleva_Status_Dword/SoftLimitMaxExceeded <-> Outputs/ToPlc/StateDWord/SoftLimitMaxExceeded
//     RulliCentroTagliTask Inputs/RULLI_CENTRO_TAGLI.Catenaria_C1_Solleva_Status_Dword/SoftLimitMinExceeded <-> Outputs/ToPlc/StateDWord/SoftLimitMinExceeded
//     RulliCentroTagliTask Inputs/RULLI_CENTRO_TAGLI.Sollevamento_C1_Act_Pos <-> Outputs/ToPlc/ActPos
//     RulliCentroTagliTask Outputs/RULLI_CENTRO_TAGLI.Catenaria_C1_Solleva.PlcToNc <-> Inputs/FromPlc
//   Galimberti/Galimberti Instance <-> NC-Task 1 SAF/Axes/C1M2
//     RulliCentroTagliTask Inputs/RULLI_CENTRO_TAGLI.Catenaria_C1_Ribalta.NcToPlc <-> Outputs/ToPlc
//     RulliCentroTagliTask Inputs/RULLI_CENTRO_TAGLI.Catenaria_C1_Ribalta_Status_Dword/CamDataQueued <-> Outputs/ToPlc/StateDWord/CamDataQueued
//     RulliCentroTagliTask Inputs/RULLI_CENTRO_TAGLI.Catenaria_C1_Ribalta_Status_Dword/CamScalingPending <-> Outputs/ToPlc/StateDWord/CamScalingPending
//     RulliCentroTagliTask Inputs/RULLI_CENTRO_TAGLI.Catenaria_C1_Ribalta_Status_Dword/CamTableQueued <-> Outputs/ToPlc/StateDWord/CamTableQueued
//     RulliCentroTagliTask Inputs/RULLI_CENTRO_TAGLI.Catenaria_C1_Ribalta_Status_Dword/CmdBuffered <-> Outputs/ToPlc/StateDWord/CmdBuffered
//     RulliCentroTagliTask Inputs/RULLI_CENTRO_TAGLI.Catenaria_C1_Ribalta_Status_Dword/Compensating <-> Outputs/ToPlc/StateDWord/Compensating
//     RulliCentroTagliTask Inputs/RULLI_CENTRO_TAGLI.Catenaria_C1_Ribalta_Status_Dword/ConstantVelocity <-> Outputs/ToPlc/StateDWord/ConstantVelocity
//     RulliCentroTagliTask Inputs/RULLI_CENTRO_TAGLI.Catenaria_C1_Ribalta_Status_Dword/ContinuousMotion <-> Outputs/ToPlc/StateDWord/ContinuousMotion
//     RulliCentroTagliTask Inputs/RULLI_CENTRO_TAGLI.Catenaria_C1_Ribalta_Status_Dword/ControlLoopClosed <-> Outputs/ToPlc/StateDWord/ControlLoopClosed
//     RulliCentroTagliTask Inputs/RULLI_CENTRO_TAGLI.Catenaria_C1_Ribalta_Status_Dword/DriveDeviceError <-> Outputs/ToPlc/StateDWord/DriveDeviceError
//     RulliCentroTagliTask Inputs/RULLI_CENTRO_TAGLI.Catenaria_C1_Ribalta_Status_Dword/Error <-> Outputs/ToPlc/StateDWord/Error
//     RulliCentroTagliTask Inputs/RULLI_CENTRO_TAGLI.Catenaria_C1_Ribalta_Status_Dword/ErrorPropagationDelayed <-> Outputs/ToPlc/StateDWord/ErrorPropagationDelayed
//     RulliCentroTagliTask Inputs/RULLI_CENTRO_TAGLI.Catenaria_C1_Ribalta_Status_Dword/ExtSetPointGenEnabled <-> Outputs/ToPlc/StateDWord/ExtSetPointGenEnabled
//     RulliCentroTagliTask Inputs/RULLI_CENTRO_TAGLI.Catenaria_C1_Ribalta_Status_Dword/ExternalLatchValid <-> Outputs/ToPlc/StateDWord/ExternalLatchValid
//     RulliCentroTagliTask Inputs/RULLI_CENTRO_TAGLI.Catenaria_C1_Ribalta_Status_Dword/HasBeenStopped <-> Outputs/ToPlc/StateDWord/HasBeenStopped
//     RulliCentroTagliTask Inputs/RULLI_CENTRO_TAGLI.Catenaria_C1_Ribalta_Status_Dword/HasJob <-> Outputs/ToPlc/StateDWord/HasJob
//     RulliCentroTagliTask Inputs/RULLI_CENTRO_TAGLI.Catenaria_C1_Ribalta_Status_Dword/Homed <-> Outputs/ToPlc/StateDWord/Homed
//     RulliCentroTagliTask Inputs/RULLI_CENTRO_TAGLI.Catenaria_C1_Ribalta_Status_Dword/HomingBusy <-> Outputs/ToPlc/StateDWord/HomingBusy
//     RulliCentroTagliTask Inputs/RULLI_CENTRO_TAGLI.Catenaria_C1_Ribalta_Status_Dword/InPositionArea <-> Outputs/ToPlc/StateDWord/InPositionArea
//     RulliCentroTagliTask Inputs/RULLI_CENTRO_TAGLI.Catenaria_C1_Ribalta_Status_Dword/InTargetPosition <-> Outputs/ToPlc/StateDWord/InTargetPosition
//     RulliCentroTagliTask Inputs/RULLI_CENTRO_TAGLI.Catenaria_C1_Ribalta_Status_Dword/IoDataInvalid <-> Outputs/ToPlc/StateDWord/IoDataInvalid
//     RulliCentroTagliTask Inputs/RULLI_CENTRO_TAGLI.Catenaria_C1_Ribalta_Status_Dword/MotionCommandsLocked <-> Outputs/ToPlc/StateDWord/MotionCommandsLocked
//     RulliCentroTagliTask Inputs/RULLI_CENTRO_TAGLI.Catenaria_C1_Ribalta_Status_Dword/NegativeDirection <-> Outputs/ToPlc/StateDWord/NegativeDirection
//     RulliCentroTagliTask Inputs/RULLI_CENTRO_TAGLI.Catenaria_C1_Ribalta_Status_Dword/NewTargetPos <-> Outputs/ToPlc/StateDWord/NewTargetPos
//     RulliCentroTagliTask Inputs/RULLI_CENTRO_TAGLI.Catenaria_C1_Ribalta_Status_Dword/NotMoving <-> Outputs/ToPlc/StateDWord/NotMoving
//     RulliCentroTagliTask Inputs/RULLI_CENTRO_TAGLI.Catenaria_C1_Ribalta_Status_Dword/Operational <-> Outputs/ToPlc/StateDWord/Operational
//     RulliCentroTagliTask Inputs/RULLI_CENTRO_TAGLI.Catenaria_C1_Ribalta_Status_Dword/PTPmode <-> Outputs/ToPlc/StateDWord/PTPmode
//     RulliCentroTagliTask Inputs/RULLI_CENTRO_TAGLI.Catenaria_C1_Ribalta_Status_Dword/PhasingActive <-> Outputs/ToPlc/StateDWord/PhasingActive
//     RulliCentroTagliTask Inputs/RULLI_CENTRO_TAGLI.Catenaria_C1_Ribalta_Status_Dword/PositiveDirection <-> Outputs/ToPlc/StateDWord/PositiveDirection
//     RulliCentroTagliTask Inputs/RULLI_CENTRO_TAGLI.Catenaria_C1_Ribalta_Status_Dword/Protected_ <-> Outputs/ToPlc/StateDWord/Protected
//     RulliCentroTagliTask Inputs/RULLI_CENTRO_TAGLI.Catenaria_C1_Ribalta_Status_Dword/SoftLimitMaxExceeded <-> Outputs/ToPlc/StateDWord/SoftLimitMaxExceeded
//     RulliCentroTagliTask Inputs/RULLI_CENTRO_TAGLI.Catenaria_C1_Ribalta_Status_Dword/SoftLimitMinExceeded <-> Outputs/ToPlc/StateDWord/SoftLimitMinExceeded
//     RulliCentroTagliTask Inputs/RULLI_CENTRO_TAGLI.Ribalta_C1_Act_Pos <-> Outputs/ToPlc/ActPos
//     RulliCentroTagliTask Outputs/RULLI_CENTRO_TAGLI.Catenaria_C1_Ribalta.PlcToNc <-> Inputs/FromPlc
//   Galimberti/Galimberti Instance <-> NC-Task 1 SAF/Axes/C1M3
//     RulliCentroTagliTask Inputs/RULLI_CENTRO_TAGLI.Catenaria_C1_Rotazione.NcToPlc <-> Outputs/ToPlc
//     RulliCentroTagliTask Inputs/RULLI_CENTRO_TAGLI.Catenaria_C1_Rotazione_Status_Dword/CamDataQueued <-> Outputs/ToPlc/StateDWord/CamDataQueued
//     RulliCentroTagliTask Inputs/RULLI_CENTRO_TAGLI.Catenaria_C1_Rotazione_Status_Dword/CamScalingPending <-> Outputs/ToPlc/StateDWord/CamScalingPending
//     RulliCentroTagliTask Inputs/RULLI_CENTRO_TAGLI.Catenaria_C1_Rotazione_Status_Dword/CamTableQueued <-> Outputs/ToPlc/StateDWord/CamTableQueued
//     RulliCentroTagliTask Inputs/RULLI_CENTRO_TAGLI.Catenaria_C1_Rotazione_Status_Dword/CmdBuffered <-> Outputs/ToPlc/StateDWord/CmdBuffered
//     RulliCentroTagliTask Inputs/RULLI_CENTRO_TAGLI.Catenaria_C1_Rotazione_Status_Dword/Compensating <-> Outputs/ToPlc/StateDWord/Compensating
//     RulliCentroTagliTask Inputs/RULLI_CENTRO_TAGLI.Catenaria_C1_Rotazione_Status_Dword/ConstantVelocity <-> Outputs/ToPlc/StateDWord/ConstantVelocity
//     RulliCentroTagliTask Inputs/RULLI_CENTRO_TAGLI.Catenaria_C1_Rotazione_Status_Dword/ContinuousMotion <-> Outputs/ToPlc/StateDWord/ContinuousMotion
//     RulliCentroTagliTask Inputs/RULLI_CENTRO_TAGLI.Catenaria_C1_Rotazione_Status_Dword/ControlLoopClosed <-> Outputs/ToPlc/StateDWord/ControlLoopClosed
//     RulliCentroTagliTask Inputs/RULLI_CENTRO_TAGLI.Catenaria_C1_Rotazione_Status_Dword/DriveDeviceError <-> Outputs/ToPlc/StateDWord/DriveDeviceError
//     RulliCentroTagliTask Inputs/RULLI_CENTRO_TAGLI.Catenaria_C1_Rotazione_Status_Dword/ErrorPropagationDelayed <-> Outputs/ToPlc/StateDWord/ErrorPropagationDelayed
//     RulliCentroTagliTask Inputs/RULLI_CENTRO_TAGLI.Catenaria_C1_Rotazione_Status_Dword/ExtSetPointGenEnabled <-> Outputs/ToPlc/StateDWord/ExtSetPointGenEnabled
//     RulliCentroTagliTask Inputs/RULLI_CENTRO_TAGLI.Catenaria_C1_Rotazione_Status_Dword/ExternalLatchValid <-> Outputs/ToPlc/StateDWord/ExternalLatchValid
//     RulliCentroTagliTask Inputs/RULLI_CENTRO_TAGLI.Catenaria_C1_Rotazione_Status_Dword/HasBeenStopped <-> Outputs/ToPlc/StateDWord/HasBeenStopped
//     RulliCentroTagliTask Inputs/RULLI_CENTRO_TAGLI.Catenaria_C1_Rotazione_Status_Dword/HasJob <-> Outputs/ToPlc/StateDWord/HasJob
//     RulliCentroTagliTask Inputs/RULLI_CENTRO_TAGLI.Catenaria_C1_Rotazione_Status_Dword/Homed <-> Outputs/ToPlc/StateDWord/Homed
//     RulliCentroTagliTask Inputs/RULLI_CENTRO_TAGLI.Catenaria_C1_Rotazione_Status_Dword/HomingBusy <-> Outputs/ToPlc/StateDWord/HomingBusy
//     RulliCentroTagliTask Inputs/RULLI_CENTRO_TAGLI.Catenaria_C1_Rotazione_Status_Dword/InPositionArea <-> Outputs/ToPlc/StateDWord/InPositionArea
//     RulliCentroTagliTask Inputs/RULLI_CENTRO_TAGLI.Catenaria_C1_Rotazione_Status_Dword/InTargetPosition <-> Outputs/ToPlc/StateDWord/InTargetPosition
//     RulliCentroTagliTask Inputs/RULLI_CENTRO_TAGLI.Catenaria_C1_Rotazione_Status_Dword/IoDataInvalid <-> Outputs/ToPlc/StateDWord/IoDataInvalid
//     RulliCentroTagliTask Inputs/RULLI_CENTRO_TAGLI.Catenaria_C1_Rotazione_Status_Dword/MotionCommandsLocked <-> Outputs/ToPlc/StateDWord/MotionCommandsLocked
//     RulliCentroTagliTask Inputs/RULLI_CENTRO_TAGLI.Catenaria_C1_Rotazione_Status_Dword/NegativeDirection <-> Outputs/ToPlc/StateDWord/NegativeDirection
//     RulliCentroTagliTask Inputs/RULLI_CENTRO_TAGLI.Catenaria_C1_Rotazione_Status_Dword/NewTargetPos <-> Outputs/ToPlc/StateDWord/NewTargetPos
//     RulliCentroTagliTask Inputs/RULLI_CENTRO_TAGLI.Catenaria_C1_Rotazione_Status_Dword/NotMoving <-> Outputs/ToPlc/StateDWord/NotMoving
//     RulliCentroTagliTask Inputs/RULLI_CENTRO_TAGLI.Catenaria_C1_Rotazione_Status_Dword/Operational <-> Outputs/ToPlc/StateDWord/Operational
//     RulliCentroTagliTask Inputs/RULLI_CENTRO_TAGLI.Catenaria_C1_Rotazione_Status_Dword/PTPmode <-> Outputs/ToPlc/StateDWord/PTPmode
//     RulliCentroTagliTask Inputs/RULLI_CENTRO_TAGLI.Catenaria_C1_Rotazione_Status_Dword/PhasingActive <-> Outputs/ToPlc/StateDWord/PhasingActive
//     RulliCentroTagliTask Inputs/RULLI_CENTRO_TAGLI.Catenaria_C1_Rotazione_Status_Dword/PositiveDirection <-> Outputs/ToPlc/StateDWord/PositiveDirection
//     RulliCentroTagliTask Inputs/RULLI_CENTRO_TAGLI.Catenaria_C1_Rotazione_Status_Dword/Protected_ <-> Outputs/ToPlc/StateDWord/Protected
//     RulliCentroTagliTask Inputs/RULLI_CENTRO_TAGLI.Catenaria_C1_Rotazione_Status_Dword/SoftLimitMaxExceeded <-> Outputs/ToPlc/StateDWord/SoftLimitMaxExceeded
//     RulliCentroTagliTask Inputs/RULLI_CENTRO_TAGLI.Catenaria_C1_Rotazione_Status_Dword/SoftLimitMinExceeded <-> Outputs/ToPlc/StateDWord/SoftLimitMinExceeded
//     RulliCentroTagliTask Outputs/RULLI_CENTRO_TAGLI.Catenaria_C1_Rotazione.PlcToNc <-> Inputs/FromPlc
//   Galimberti/Galimberti Instance <-> NC-Task 1 SAF/Axes/C2M1
//     RulliCentroTagliTask Inputs/RULLI_CENTRO_TAGLI.Catenaria_C2_Rotazione.NcToPlc <-> Outputs/ToPlc
//     RulliCentroTagliTask Inputs/RULLI_CENTRO_TAGLI.Catenaria_C2_Rotazione_Status_Dword/CamDataQueued <-> Outputs/ToPlc/StateDWord/CamDataQueued
//     RulliCentroTagliTask Inputs/RULLI_CENTRO_TAGLI.Catenaria_C2_Rotazione_Status_Dword/CamScalingPending <-> Outputs/ToPlc/StateDWord/CamScalingPending
//     RulliCentroTagliTask Inputs/RULLI_CENTRO_TAGLI.Catenaria_C2_Rotazione_Status_Dword/CamTableQueued <-> Outputs/ToPlc/StateDWord/CamTableQueued
//     RulliCentroTagliTask Inputs/RULLI_CENTRO_TAGLI.Catenaria_C2_Rotazione_Status_Dword/CmdBuffered <-> Outputs/ToPlc/StateDWord/CmdBuffered
//     RulliCentroTagliTask Inputs/RULLI_CENTRO_TAGLI.Catenaria_C2_Rotazione_Status_Dword/Compensating <-> Outputs/ToPlc/StateDWord/Compensating
//     RulliCentroTagliTask Inputs/RULLI_CENTRO_TAGLI.Catenaria_C2_Rotazione_Status_Dword/ConstantVelocity <-> Outputs/ToPlc/StateDWord/ConstantVelocity
//     RulliCentroTagliTask Inputs/RULLI_CENTRO_TAGLI.Catenaria_C2_Rotazione_Status_Dword/ContinuousMotion <-> Outputs/ToPlc/StateDWord/ContinuousMotion
//     RulliCentroTagliTask Inputs/RULLI_CENTRO_TAGLI.Catenaria_C2_Rotazione_Status_Dword/ControlLoopClosed <-> Outputs/ToPlc/StateDWord/ControlLoopClosed
//     RulliCentroTagliTask Inputs/RULLI_CENTRO_TAGLI.Catenaria_C2_Rotazione_Status_Dword/DriveDeviceError <-> Outputs/ToPlc/StateDWord/DriveDeviceError
//     RulliCentroTagliTask Inputs/RULLI_CENTRO_TAGLI.Catenaria_C2_Rotazione_Status_Dword/ErrorPropagationDelayed <-> Outputs/ToPlc/StateDWord/ErrorPropagationDelayed
//     RulliCentroTagliTask Inputs/RULLI_CENTRO_TAGLI.Catenaria_C2_Rotazione_Status_Dword/ExtSetPointGenEnabled <-> Outputs/ToPlc/StateDWord/ExtSetPointGenEnabled
//     RulliCentroTagliTask Inputs/RULLI_CENTRO_TAGLI.Catenaria_C2_Rotazione_Status_Dword/ExternalLatchValid <-> Outputs/ToPlc/StateDWord/ExternalLatchValid
//     RulliCentroTagliTask Inputs/RULLI_CENTRO_TAGLI.Catenaria_C2_Rotazione_Status_Dword/HasBeenStopped <-> Outputs/ToPlc/StateDWord/HasBeenStopped
//     RulliCentroTagliTask Inputs/RULLI_CENTRO_TAGLI.Catenaria_C2_Rotazione_Status_Dword/HasJob <-> Outputs/ToPlc/StateDWord/HasJob
//     RulliCentroTagliTask Inputs/RULLI_CENTRO_TAGLI.Catenaria_C2_Rotazione_Status_Dword/Homed <-> Outputs/ToPlc/StateDWord/Homed
//     RulliCentroTagliTask Inputs/RULLI_CENTRO_TAGLI.Catenaria_C2_Rotazione_Status_Dword/HomingBusy <-> Outputs/ToPlc/StateDWord/HomingBusy
//     RulliCentroTagliTask Inputs/RULLI_CENTRO_TAGLI.Catenaria_C2_Rotazione_Status_Dword/InPositionArea <-> Outputs/ToPlc/StateDWord/InPositionArea
//     RulliCentroTagliTask Inputs/RULLI_CENTRO_TAGLI.Catenaria_C2_Rotazione_Status_Dword/InTargetPosition <-> Outputs/ToPlc/StateDWord/InTargetPosition
//     RulliCentroTagliTask Inputs/RULLI_CENTRO_TAGLI.Catenaria_C2_Rotazione_Status_Dword/IoDataInvalid <-> Outputs/ToPlc/StateDWord/IoDataInvalid
//     RulliCentroTagliTask Inputs/RULLI_CENTRO_TAGLI.Catenaria_C2_Rotazione_Status_Dword/MotionCommandsLocked <-> Outputs/ToPlc/StateDWord/MotionCommandsLocked
//     RulliCentroTagliTask Inputs/RULLI_CENTRO_TAGLI.Catenaria_C2_Rotazione_Status_Dword/NegativeDirection <-> Outputs/ToPlc/StateDWord/NegativeDirection
//     RulliCentroTagliTask Inputs/RULLI_CENTRO_TAGLI.Catenaria_C2_Rotazione_Status_Dword/NewTargetPos <-> Outputs/ToPlc/StateDWord/NewTargetPos
//     RulliCentroTagliTask Inputs/RULLI_CENTRO_TAGLI.Catenaria_C2_Rotazione_Status_Dword/NotMoving <-> Outputs/ToPlc/StateDWord/NotMoving
//     RulliCentroTagliTask Inputs/RULLI_CENTRO_TAGLI.Catenaria_C2_Rotazione_Status_Dword/Operational <-> Outputs/ToPlc/StateDWord/Operational
//     RulliCentroTagliTask Inputs/RULLI_CENTRO_TAGLI.Catenaria_C2_Rotazione_Status_Dword/PTPmode <-> Outputs/ToPlc/StateDWord/PTPmode
//     RulliCentroTagliTask Inputs/RULLI_CENTRO_TAGLI.Catenaria_C2_Rotazione_Status_Dword/PhasingActive <-> Outputs/ToPlc/StateDWord/PhasingActive
//     RulliCentroTagliTask Inputs/RULLI_CENTRO_TAGLI.Catenaria_C2_Rotazione_Status_Dword/PositiveDirection <-> Outputs/ToPlc/StateDWord/PositiveDirection
//     RulliCentroTagliTask Inputs/RULLI_CENTRO_TAGLI.Catenaria_C2_Rotazione_Status_Dword/Protected_ <-> Outputs/ToPlc/StateDWord/Protected
//     RulliCentroTagliTask Inputs/RULLI_CENTRO_TAGLI.Catenaria_C2_Rotazione_Status_Dword/SoftLimitMaxExceeded <-> Outputs/ToPlc/StateDWord/SoftLimitMaxExceeded
//     RulliCentroTagliTask Inputs/RULLI_CENTRO_TAGLI.Catenaria_C2_Rotazione_Status_Dword/SoftLimitMinExceeded <-> Outputs/ToPlc/StateDWord/SoftLimitMinExceeded
//     RulliCentroTagliTask Outputs/RULLI_CENTRO_TAGLI.Catenaria_C2_Rotazione.PlcToNc <-> Inputs/FromPlc
//   Galimberti/Galimberti Instance <-> NC-Task 1 SAF/Axes/C3
//     RulliCentroTagliTask Inputs/RULLI_CENTRO_TAGLI.Catenaria_C3_Rotazione.NcToPlc <-> Outputs/ToPlc
//     RulliCentroTagliTask Inputs/RULLI_CENTRO_TAGLI.Catenaria_C3_Rotazione_Status_Dword/CamDataQueued <-> Outputs/ToPlc/StateDWord/CamDataQueued
//     RulliCentroTagliTask Inputs/RULLI_CENTRO_TAGLI.Catenaria_C3_Rotazione_Status_Dword/CamScalingPending <-> Outputs/ToPlc/StateDWord/CamScalingPending
//     RulliCentroTagliTask Inputs/RULLI_CENTRO_TAGLI.Catenaria_C3_Rotazione_Status_Dword/CamTableQueued <-> Outputs/ToPlc/StateDWord/CamTableQueued
//     RulliCentroTagliTask Inputs/RULLI_CENTRO_TAGLI.Catenaria_C3_Rotazione_Status_Dword/CmdBuffered <-> Outputs/ToPlc/StateDWord/CmdBuffered
//     RulliCentroTagliTask Inputs/RULLI_CENTRO_TAGLI.Catenaria_C3_Rotazione_Status_Dword/Compensating <-> Outputs/ToPlc/StateDWord/Compensating
//     RulliCentroTagliTask Inputs/RULLI_CENTRO_TAGLI.Catenaria_C3_Rotazione_Status_Dword/ConstantVelocity <-> Outputs/ToPlc/StateDWord/ConstantVelocity
//     RulliCentroTagliTask Inputs/RULLI_CENTRO_TAGLI.Catenaria_C3_Rotazione_Status_Dword/ContinuousMotion <-> Outputs/ToPlc/StateDWord/ContinuousMotion
//     RulliCentroTagliTask Inputs/RULLI_CENTRO_TAGLI.Catenaria_C3_Rotazione_Status_Dword/ControlLoopClosed <-> Outputs/ToPlc/StateDWord/ControlLoopClosed
//     RulliCentroTagliTask Inputs/RULLI_CENTRO_TAGLI.Catenaria_C3_Rotazione_Status_Dword/DriveDeviceError <-> Outputs/ToPlc/StateDWord/DriveDeviceError
//     RulliCentroTagliTask Inputs/RULLI_CENTRO_TAGLI.Catenaria_C3_Rotazione_Status_Dword/ErrorPropagationDelayed <-> Outputs/ToPlc/StateDWord/ErrorPropagationDelayed
//     RulliCentroTagliTask Inputs/RULLI_CENTRO_TAGLI.Catenaria_C3_Rotazione_Status_Dword/ExtSetPointGenEnabled <-> Outputs/ToPlc/StateDWord/ExtSetPointGenEnabled
//     RulliCentroTagliTask Inputs/RULLI_CENTRO_TAGLI.Catenaria_C3_Rotazione_Status_Dword/ExternalLatchValid <-> Outputs/ToPlc/StateDWord/ExternalLatchValid
//     RulliCentroTagliTask Inputs/RULLI_CENTRO_TAGLI.Catenaria_C3_Rotazione_Status_Dword/HasBeenStopped <-> Outputs/ToPlc/StateDWord/HasBeenStopped
//     RulliCentroTagliTask Inputs/RULLI_CENTRO_TAGLI.Catenaria_C3_Rotazione_Status_Dword/HasJob <-> Outputs/ToPlc/StateDWord/HasJob
//     RulliCentroTagliTask Inputs/RULLI_CENTRO_TAGLI.Catenaria_C3_Rotazione_Status_Dword/Homed <-> Outputs/ToPlc/StateDWord/Homed
//     RulliCentroTagliTask Inputs/RULLI_CENTRO_TAGLI.Catenaria_C3_Rotazione_Status_Dword/HomingBusy <-> Outputs/ToPlc/StateDWord/HomingBusy
//     RulliCentroTagliTask Inputs/RULLI_CENTRO_TAGLI.Catenaria_C3_Rotazione_Status_Dword/InPositionArea <-> Outputs/ToPlc/StateDWord/InPositionArea
//     RulliCentroTagliTask Inputs/RULLI_CENTRO_TAGLI.Catenaria_C3_Rotazione_Status_Dword/InTargetPosition <-> Outputs/ToPlc/StateDWord/InTargetPosition
//     RulliCentroTagliTask Inputs/RULLI_CENTRO_TAGLI.Catenaria_C3_Rotazione_Status_Dword/IoDataInvalid <-> Outputs/ToPlc/StateDWord/IoDataInvalid
//     RulliCentroTagliTask Inputs/RULLI_CENTRO_TAGLI.Catenaria_C3_Rotazione_Status_Dword/MotionCommandsLocked <-> Outputs/ToPlc/StateDWord/MotionCommandsLocked
//     RulliCentroTagliTask Inputs/RULLI_CENTRO_TAGLI.Catenaria_C3_Rotazione_Status_Dword/NegativeDirection <-> Outputs/ToPlc/StateDWord/NegativeDirection
//     RulliCentroTagliTask Inputs/RULLI_CENTRO_TAGLI.Catenaria_C3_Rotazione_Status_Dword/NewTargetPos <-> Outputs/ToPlc/StateDWord/NewTargetPos
//     RulliCentroTagliTask Inputs/RULLI_CENTRO_TAGLI.Catenaria_C3_Rotazione_Status_Dword/NotMoving <-> Outputs/ToPlc/StateDWord/NotMoving
//     RulliCentroTagliTask Inputs/RULLI_CENTRO_TAGLI.Catenaria_C3_Rotazione_Status_Dword/Operational <-> Outputs/ToPlc/StateDWord/Operational
//     RulliCentroTagliTask Inputs/RULLI_CENTRO_TAGLI.Catenaria_C3_Rotazione_Status_Dword/PTPmode <-> Outputs/ToPlc/StateDWord/PTPmode
//     RulliCentroTagliTask Inputs/RULLI_CENTRO_TAGLI.Catenaria_C3_Rotazione_Status_Dword/PhasingActive <-> Outputs/ToPlc/StateDWord/PhasingActive
//     RulliCentroTagliTask Inputs/RULLI_CENTRO_TAGLI.Catenaria_C3_Rotazione_Status_Dword/PositiveDirection <-> Outputs/ToPlc/StateDWord/PositiveDirection
//     RulliCentroTagliTask Inputs/RULLI_CENTRO_TAGLI.Catenaria_C3_Rotazione_Status_Dword/Protected_ <-> Outputs/ToPlc/StateDWord/Protected
//     RulliCentroTagliTask Inputs/RULLI_CENTRO_TAGLI.Catenaria_C3_Rotazione_Status_Dword/SoftLimitMaxExceeded <-> Outputs/ToPlc/StateDWord/SoftLimitMaxExceeded
//     RulliCentroTagliTask Inputs/RULLI_CENTRO_TAGLI.Catenaria_C3_Rotazione_Status_Dword/SoftLimitMinExceeded <-> Outputs/ToPlc/StateDWord/SoftLimitMinExceeded
//     RulliCentroTagliTask Outputs/RULLI_CENTRO_TAGLI.Catenaria_C3_Rotazione.PlcToNc <-> Inputs/FromPlc
//   Galimberti/Galimberti Instance <-> NC-Task 1 SAF/Axes/C4
//     RulliCentroTagliTask Inputs/RULLI_CENTRO_TAGLI.Catenaria_C4_Rotazione.NcToPlc <-> Outputs/ToPlc
//     RulliCentroTagliTask Inputs/RULLI_CENTRO_TAGLI.Catenaria_C4_Rotazione_Status_Dword/CamDataQueued <-> Outputs/ToPlc/StateDWord/CamDataQueued
//     RulliCentroTagliTask Inputs/RULLI_CENTRO_TAGLI.Catenaria_C4_Rotazione_Status_Dword/CamScalingPending <-> Outputs/ToPlc/StateDWord/CamScalingPending
//     RulliCentroTagliTask Inputs/RULLI_CENTRO_TAGLI.Catenaria_C4_Rotazione_Status_Dword/CamTableQueued <-> Outputs/ToPlc/StateDWord/CamTableQueued
//     RulliCentroTagliTask Inputs/RULLI_CENTRO_TAGLI.Catenaria_C4_Rotazione_Status_Dword/CmdBuffered <-> Outputs/ToPlc/StateDWord/CmdBuffered
//     RulliCentroTagliTask Inputs/RULLI_CENTRO_TAGLI.Catenaria_C4_Rotazione_Status_Dword/Compensating <-> Outputs/ToPlc/StateDWord/Compensating
//     RulliCentroTagliTask Inputs/RULLI_CENTRO_TAGLI.Catenaria_C4_Rotazione_Status_Dword/ConstantVelocity <-> Outputs/ToPlc/StateDWord/ConstantVelocity
//     RulliCentroTagliTask Inputs/RULLI_CENTRO_TAGLI.Catenaria_C4_Rotazione_Status_Dword/ContinuousMotion <-> Outputs/ToPlc/StateDWord/ContinuousMotion
//     RulliCentroTagliTask Inputs/RULLI_CENTRO_TAGLI.Catenaria_C4_Rotazione_Status_Dword/ControlLoopClosed <-> Outputs/ToPlc/StateDWord/ControlLoopClosed
//     RulliCentroTagliTask Inputs/RULLI_CENTRO_TAGLI.Catenaria_C4_Rotazione_Status_Dword/DriveDeviceError <-> Outputs/ToPlc/StateDWord/DriveDeviceError
//     RulliCentroTagliTask Inputs/RULLI_CENTRO_TAGLI.Catenaria_C4_Rotazione_Status_Dword/Error <-> Outputs/ToPlc/StateDWord/Error
//     RulliCentroTagliTask Inputs/RULLI_CENTRO_TAGLI.Catenaria_C4_Rotazione_Status_Dword/ErrorPropagationDelayed <-> Outputs/ToPlc/StateDWord/ErrorPropagationDelayed
//     RulliCentroTagliTask Inputs/RULLI_CENTRO_TAGLI.Catenaria_C4_Rotazione_Status_Dword/ExtSetPointGenEnabled <-> Outputs/ToPlc/StateDWord/ExtSetPointGenEnabled
//     RulliCentroTagliTask Inputs/RULLI_CENTRO_TAGLI.Catenaria_C4_Rotazione_Status_Dword/ExternalLatchValid <-> Outputs/ToPlc/StateDWord/ExternalLatchValid
//     RulliCentroTagliTask Inputs/RULLI_CENTRO_TAGLI.Catenaria_C4_Rotazione_Status_Dword/HasBeenStopped <-> Outputs/ToPlc/StateDWord/HasBeenStopped
//     RulliCentroTagliTask Inputs/RULLI_CENTRO_TAGLI.Catenaria_C4_Rotazione_Status_Dword/HasJob <-> Outputs/ToPlc/StateDWord/HasJob
//     RulliCentroTagliTask Inputs/RULLI_CENTRO_TAGLI.Catenaria_C4_Rotazione_Status_Dword/Homed <-> Outputs/ToPlc/StateDWord/Homed
//     RulliCentroTagliTask Inputs/RULLI_CENTRO_TAGLI.Catenaria_C4_Rotazione_Status_Dword/HomingBusy <-> Outputs/ToPlc/StateDWord/HomingBusy
//     RulliCentroTagliTask Inputs/RULLI_CENTRO_TAGLI.Catenaria_C4_Rotazione_Status_Dword/InPositionArea <-> Outputs/ToPlc/StateDWord/InPositionArea
